// ---- POUs/BACnet_FBCode/FB_BACnet_SCSII_2_GRAHA_ENERGY.TcPOU
(* Usage : 
fbSCSII_2_GRAHA_ENERGY : FB_BACnet_SCSII_2_GRAHA_ENERGY :=(Client:=(nDeviceInstance := 356)); 
*)
FUNCTION_BLOCK  FB_BACnet_SCSII_2_GRAHA_ENERGY
VAR_INPUT CONSTANT
	Client : FB_BACnet_Client := (tReadCycleTime:=T#10S,nMaxParallelRequests:=20);
	SCSII_2_GRAHA_ENERGY: FB_BACnetRM_Device := (Client:=Client);
	Exhaust_Fan_GF_1_ST: FB_BACnetRM_BI := (Client:=Client,nObjectInstance:=208);
	Exhaust_Fan_GF_1_TR: FB_BACnetRM_BI := (Client:=Client,nObjectInstance:=209);
	Exhaust_Fan_GF_2_ST: FB_BACnetRM_BI := (Client:=Client,nObjectInstance:=210);
	Exhaust_Fan_GF_2_TR: FB_BACnetRM_BI := (Client:=Client,nObjectInstance:=211);
	Exhaust_Fan_GF_3_ST: FB_BACnetRM_BI := (Client:=Client,nObjectInstance:=212);
	Exhaust_Fan_GF_3_TR: FB_BACnetRM_BI := (Client:=Client,nObjectInstance:=213);
	Intake_Fan_GF_1_ST: FB_BACnetRM_BI := (Client:=Client,nObjectInstance:=214);
	Intake_Fan_GF_1_TR: FB_BACnetRM_BI := (Client:=Client,nObjectInstance:=215);
	Intake_Fan_GF_2_ST: FB_BACnetRM_BI := (Client:=Client,nObjectInstance:=216);
	Intake_Fan_GF_2_TR: FB_BACnetRM_BI := (Client:=Client,nObjectInstance:=217);
	Toilet_Exh_Fan_GF_1_ST: FB_BACnetRM_BI := (Client:=Client,nObjectInstance:=218);
	Toilet_Exh_Fan_GF_1_TR: FB_BACnetRM_BI := (Client:=Client,nObjectInstance:=219);
	Exhaust_Fan_MZ_1_ST: FB_BACnetRM_BI := (Client:=Client,nObjectInstance:=220);
	Exhaust_Fan_MZ_1_TR: FB_BACnetRM_BI := (Client:=Client,nObjectInstance:=221);
	Exhaust_Fan_MZ_2_ST: FB_BACnetRM_BI := (Client:=Client,nObjectInstance:=222);
	Exhaust_Fan_MZ_2_TR: FB_BACnetRM_BI := (Client:=Client,nObjectInstance:=223);
	Exhaust_Fan_MZ_3_ST: FB_BACnetRM_BI := (Client:=Client,nObjectInstance:=224);
	Exhaust_Fan_MZ_3_TR: FB_BACnetRM_BI := (Client:=Client,nObjectInstance:=225);
	Exhaust_Fan_MZ_4_ST: FB_BACnetRM_BI := (Client:=Client,nObjectInstance:=226);
	Exhaust_Fan_MZ_4_TR: FB_BACnetRM_BI := (Client:=Client,nObjectInstance:=227);
	Exhaust_Fan_MZ_5_ST: FB_BACnetRM_BI := (Client:=Client,nObjectInstance:=228);
	Exhaust_Fan_MZ_5_TR: FB_BACnetRM_BI := (Client:=Client,nObjectInstance:=229);
	Exhaust_Fan_MZ_6_ST: FB_BACnetRM_BI := (Client:=Client,nObjectInstance:=230);
	Exhaust_Fan_MZ_6_TR: FB_BACnetRM_BI := (Client:=Client,nObjectInstance:=231);
	Exhaust_Fan_MZ_7_ST: FB_BACnetRM_BI := (Client:=Client,nObjectInstance:=232);
	Exhaust_Fan_MZ_7_TR: FB_BACnetRM_BI := (Client:=Client,nObjectInstance:=233);
	Intake_Fan_MZ_1_ST: FB_BACnetRM_BI := (Client:=Client,nObjectInstance:=234);
	Intake_Fan_MZ_1_TR: FB_BACnetRM_BI := (Client:=Client,nObjectInstance:=235);
	Toilet_Exh_Fan_MZ_1_ST: FB_BACnetRM_BI := (Client:=Client,nObjectInstance:=236);
	Toilet_Exh_Fan_MZ_1_TR: FB_BACnetRM_BI := (Client:=Client,nObjectInstance:=237);
	Exhaust_Fan_2_1_ST: FB_BACnetRM_BI := (Client:=Client,nObjectInstance:=238);
	Exhaust_Fan_2_1_TR: FB_BACnetRM_BI := (Client:=Client,nObjectInstance:=239);
	Exhaust_Fan_2_2_ST: FB_BACnetRM_BI := (Client:=Client,nObjectInstance:=240);
	Exhaust_Fan_2_2_TR: FB_BACnetRM_BI := (Client:=Client,nObjectInstance:=241);
	Exhaust_Fan_2_3_ST: FB_BACnetRM_BI := (Client:=Client,nObjectInstance:=242);
	Exhaust_Fan_2_3_TR: FB_BACnetRM_BI := (Client:=Client,nObjectInstance:=243);
	Exhaust_Fan_2_4_ST: FB_BACnetRM_BI := (Client:=Client,nObjectInstance:=244);
	Exhaust_Fan_2_4_TR: FB_BACnetRM_BI := (Client:=Client,nObjectInstance:=245);
	Intake_Fan_2_1_ST: FB_BACnetRM_BI := (Client:=Client,nObjectInstance:=246);
	Intake_Fan_2_1_TR: FB_BACnetRM_BI := (Client:=Client,nObjectInstance:=247);
	Intake_Fan_2_2_ST: FB_BACnetRM_BI := (Client:=Client,nObjectInstance:=248);
	Intake_Fan_2_2_TR: FB_BACnetRM_BI := (Client:=Client,nObjectInstance:=249);
	Intake_Fan_2_3_ST: FB_BACnetRM_BI := (Client:=Client,nObjectInstance:=250);
	Intake_Fan_2_3_TR: FB_BACnetRM_BI := (Client:=Client,nObjectInstance:=251);
	Toilet_Exh_Fan_2_1_ST: FB_BACnetRM_BI := (Client:=Client,nObjectInstance:=252);
	Toilet_Exh_Fan_2_1_TR: FB_BACnetRM_BI := (Client:=Client,nObjectInstance:=253);
	Intake_Fan_4_1_ST: FB_BACnetRM_BI := (Client:=Client,nObjectInstance:=254);
	Intake_Fan_4_1_TR: FB_BACnetRM_BI := (Client:=Client,nObjectInstance:=255);
	Intake_Fan_4_2_ST: FB_BACnetRM_BI := (Client:=Client,nObjectInstance:=256);
	Intake_Fan_4_2_TR: FB_BACnetRM_BI := (Client:=Client,nObjectInstance:=257);
	Intake_Fan_4_3_ST: FB_BACnetRM_BI := (Client:=Client,nObjectInstance:=258);
	Intake_Fan_4_3_TR: FB_BACnetRM_BI := (Client:=Client,nObjectInstance:=259);
	Exhaust_Fan_4_5_ST: FB_BACnetRM_BI := (Client:=Client,nObjectInstance:=260);
	Exhaust_Fan_4_5_TR: FB_BACnetRM_BI := (Client:=Client,nObjectInstance:=261);
	Exhaust_Fan_4_6_ST: FB_BACnetRM_BI := (Client:=Client,nObjectInstance:=262);
	Exhaust_Fan_4_6_TR: FB_BACnetRM_BI := (Client:=Client,nObjectInstance:=263);
	Exhaust_Fan_4_7_ST: FB_BACnetRM_BI := (Client:=Client,nObjectInstance:=264);
	Exhaust_Fan_4_7_TR: FB_BACnetRM_BI := (Client:=Client,nObjectInstance:=265);
	Exhaust_Fan_3_7_ST: FB_BACnetRM_BI := (Client:=Client,nObjectInstance:=266);
	Exhaust_Fan_3_7_TR: FB_BACnetRM_BI := (Client:=Client,nObjectInstance:=267);
	Intake_Fan_3_1_ST: FB_BACnetRM_BI := (Client:=Client,nObjectInstance:=268);
	General_Fire_Alm: FB_BACnetRM_BI := (Client:=Client,nObjectInstance:=269);
	Intake_Fan_3_2_ST: FB_BACnetRM_BI := (Client:=Client,nObjectInstance:=270);
	Intake_Fan_3_2_TR: FB_BACnetRM_BI := (Client:=Client,nObjectInstance:=271);
	Exhaust_Fan_B5_1_ST: FB_BACnetRM_BI := (Client:=Client,nObjectInstance:=470);
	Exhaust_Fan_B5_2_ST: FB_BACnetRM_BI := (Client:=Client,nObjectInstance:=471);
	Exhaust_Fan_B5_3_ST: FB_BACnetRM_BI := (Client:=Client,nObjectInstance:=472);
	Intake_Fan_B5_1_ST: FB_BACnetRM_BI := (Client:=Client,nObjectInstance:=473);
	Intake_Fan_B5_2_ST: FB_BACnetRM_BI := (Client:=Client,nObjectInstance:=474);
	Intake_Fan_B5_3_ST: FB_BACnetRM_BI := (Client:=Client,nObjectInstance:=475);
	Spare_1_ST: FB_BACnetRM_BI := (Client:=Client,nObjectInstance:=476);
	Spare_2_ST: FB_BACnetRM_BI := (Client:=Client,nObjectInstance:=477);
	Exhaust_Fan_B5_1_TR: FB_BACnetRM_BI := (Client:=Client,nObjectInstance:=478);
	Exhaust_Fan_B5_2_TR: FB_BACnetRM_BI := (Client:=Client,nObjectInstance:=479);
	Exhaust_Fan_B5_3_TR: FB_BACnetRM_BI := (Client:=Client,nObjectInstance:=480);
	Intake_Fan_B5_1_TR: FB_BACnetRM_BI := (Client:=Client,nObjectInstance:=481);
	Intake_Fan_B5_2_TR: FB_BACnetRM_BI := (Client:=Client,nObjectInstance:=482);
	Intake_Fan_B5_3_TR: FB_BACnetRM_BI := (Client:=Client,nObjectInstance:=483);
	Spare_1_TR: FB_BACnetRM_BI := (Client:=Client,nObjectInstance:=484);
	Spare_2_TR: FB_BACnetRM_BI := (Client:=Client,nObjectInstance:=485);
	Exhaust_Fan_B4_1_ST: FB_BACnetRM_BI := (Client:=Client,nObjectInstance:=486);
	Exhaust_Fan_B4_2_ST: FB_BACnetRM_BI := (Client:=Client,nObjectInstance:=487);
	Exhaust_Fan_B4_3_ST: FB_BACnetRM_BI := (Client:=Client,nObjectInstance:=488);
	Intake_Fan_B4_1_ST: FB_BACnetRM_BI := (Client:=Client,nObjectInstance:=489);
	Intake_Fan_B4_2_ST: FB_BACnetRM_BI := (Client:=Client,nObjectInstance:=490);
	Intake_Fan_B4_3_ST: FB_BACnetRM_BI := (Client:=Client,nObjectInstance:=491);
	Spare_1_ST_X: FB_BACnetRM_BI := (Client:=Client,nObjectInstance:=492);
	Spare_2_ST_X: FB_BACnetRM_BI := (Client:=Client,nObjectInstance:=493);
	Exhaust_Fan_B4_1_TR: FB_BACnetRM_BI := (Client:=Client,nObjectInstance:=494);
	Exhaust_Fan_B4_2_TR: FB_BACnetRM_BI := (Client:=Client,nObjectInstance:=495);
	Exhaust_Fan_B4_3_TR: FB_BACnetRM_BI := (Client:=Client,nObjectInstance:=496);
	Intake_Fan_B4_1_TR: FB_BACnetRM_BI := (Client:=Client,nObjectInstance:=497);
	Intake_Fan_B4_2_TR: FB_BACnetRM_BI := (Client:=Client,nObjectInstance:=498);
	Intake_Fan_B4_3_TR: FB_BACnetRM_BI := (Client:=Client,nObjectInstance:=499);
	Spare_1_TR_X: FB_BACnetRM_BI := (Client:=Client,nObjectInstance:=500);
	Spare_2_TR_X: FB_BACnetRM_BI := (Client:=Client,nObjectInstance:=501);
	Exhaust_Fan_B3_1_ST: FB_BACnetRM_BI := (Client:=Client,nObjectInstance:=502);
	Exhaust_Fan_B3_2_ST: FB_BACnetRM_BI := (Client:=Client,nObjectInstance:=503);
	Exhaust_Fan_B3_3_ST: FB_BACnetRM_BI := (Client:=Client,nObjectInstance:=504);
	Intake_Fan_B3_1_ST: FB_BACnetRM_BI := (Client:=Client,nObjectInstance:=505);
	Intake_Fan_B3_2_ST: FB_BACnetRM_BI := (Client:=Client,nObjectInstance:=506);
	Intake_Fan_B3_3_ST: FB_BACnetRM_BI := (Client:=Client,nObjectInstance:=507);
	Spare_1_ST_X_X: FB_BACnetRM_BI := (Client:=Client,nObjectInstance:=508);
	Spare_2_ST_X_X: FB_BACnetRM_BI := (Client:=Client,nObjectInstance:=509);
	Exhaust_Fan_B3_1_TR: FB_BACnetRM_BI := (Client:=Client,nObjectInstance:=510);
	Exhaust_Fan_B3_2_TR: FB_BACnetRM_BI := (Client:=Client,nObjectInstance:=511);
	Exhaust_Fan_B3_3_TR: FB_BACnetRM_BI := (Client:=Client,nObjectInstance:=512);
	Intake_Fan_B3_1_TR: FB_BACnetRM_BI := (Client:=Client,nObjectInstance:=513);
	Intake_Fan_B3_2_TR: FB_BACnetRM_BI := (Client:=Client,nObjectInstance:=514);
	Intake_Fan_B3_3_TR: FB_BACnetRM_BI := (Client:=Client,nObjectInstance:=515);
	Spare_1_TR_X_X: FB_BACnetRM_BI := (Client:=Client,nObjectInstance:=516);
	Spare_2_TR_X_X: FB_BACnetRM_BI := (Client:=Client,nObjectInstance:=517);
	Exhaust_Fan_B2_1_ST: FB_BACnetRM_BI := (Client:=Client,nObjectInstance:=518);
	Exhaust_Fan_B2_2_ST: FB_BACnetRM_BI := (Client:=Client,nObjectInstance:=519);
	Exhaust_Fan_B2_3_ST: FB_BACnetRM_BI := (Client:=Client,nObjectInstance:=520);
	Intake_Fan_B2_1_ST: FB_BACnetRM_BI := (Client:=Client,nObjectInstance:=521);
	Intake_Fan_B2_2_ST: FB_BACnetRM_BI := (Client:=Client,nObjectInstance:=522);
	Intake_Fan_B2_3_ST: FB_BACnetRM_BI := (Client:=Client,nObjectInstance:=523);
	Reset_Alarm_Fire_Pump_S: FB_BACnetRM_BI := (Client:=Client,nObjectInstance:=524);
	Spare_2_ST_X_X_X: FB_BACnetRM_BI := (Client:=Client,nObjectInstance:=525);
	Exhaust_Fan_B2_1_TR: FB_BACnetRM_BI := (Client:=Client,nObjectInstance:=526);
	Exhaust_Fan_B2_2_TR: FB_BACnetRM_BI := (Client:=Client,nObjectInstance:=527);
	Exhaust_Fan_B2_3_TR: FB_BACnetRM_BI := (Client:=Client,nObjectInstance:=528);
	Intake_Fan_B2_1_TR: FB_BACnetRM_BI := (Client:=Client,nObjectInstance:=529);
	Intake_Fan_B2_2_TR: FB_BACnetRM_BI := (Client:=Client,nObjectInstance:=530);
	Intake_Fan_B2_3_TR: FB_BACnetRM_BI := (Client:=Client,nObjectInstance:=531);
	Spare_1_TR_X_X_X: FB_BACnetRM_BI := (Client:=Client,nObjectInstance:=532);
	Spare_2_TR_X_X_X: FB_BACnetRM_BI := (Client:=Client,nObjectInstance:=533);
	Exhaust_Fan_B1_1_ST: FB_BACnetRM_BI := (Client:=Client,nObjectInstance:=534);
	Exhaust_Fan_B1_2_ST: FB_BACnetRM_BI := (Client:=Client,nObjectInstance:=535);
	Exhaust_Fan_B1_3_ST: FB_BACnetRM_BI := (Client:=Client,nObjectInstance:=536);
	Intake_Fan_B1_1_ST: FB_BACnetRM_BI := (Client:=Client,nObjectInstance:=537);
	Intake_Fan_B1_2_ST: FB_BACnetRM_BI := (Client:=Client,nObjectInstance:=538);
	Intake_Fan_B1_3_ST: FB_BACnetRM_BI := (Client:=Client,nObjectInstance:=539);
	Spare_1_ST_X_X_X: FB_BACnetRM_BI := (Client:=Client,nObjectInstance:=540);
	Spare_2_ST_X_X_X_X: FB_BACnetRM_BI := (Client:=Client,nObjectInstance:=541);
	Exhaust_Fan_B1_1_TR: FB_BACnetRM_BI := (Client:=Client,nObjectInstance:=542);
	Exhaust_Fan_B1_2_TR: FB_BACnetRM_BI := (Client:=Client,nObjectInstance:=543);
	Exhaust_Fan_B1_3_TR: FB_BACnetRM_BI := (Client:=Client,nObjectInstance:=544);
	Intake_Fan_B1_1_TR: FB_BACnetRM_BI := (Client:=Client,nObjectInstance:=545);
	Intake_Fan_B1_2_TR: FB_BACnetRM_BI := (Client:=Client,nObjectInstance:=546);
	Intake_Fan_B1_3_TR: FB_BACnetRM_BI := (Client:=Client,nObjectInstance:=547);
	Spare_1_TR_X_X_X_X: FB_BACnetRM_BI := (Client:=Client,nObjectInstance:=548);
	Spare_2_TR_X_X_X_X: FB_BACnetRM_BI := (Client:=Client,nObjectInstance:=549);
	Intake_Fan_3_3_ST: FB_BACnetRM_BI := (Client:=Client,nObjectInstance:=599);
	Intake_Fan_3_3_TR: FB_BACnetRM_BI := (Client:=Client,nObjectInstance:=600);
	Toilet_Exh_Fan_3_1_ST: FB_BACnetRM_BI := (Client:=Client,nObjectInstance:=601);
	Toilet_Exh_Fan_3_1_TR: FB_BACnetRM_BI := (Client:=Client,nObjectInstance:=602);
	Exh_Fan_Mech_2_1_ST: FB_BACnetRM_BI := (Client:=Client,nObjectInstance:=603);
	Exh_Fan_Mech_2_2_ST: FB_BACnetRM_BI := (Client:=Client,nObjectInstance:=604);
	Exh_Fan_Mech_2_1_TR: FB_BACnetRM_BI := (Client:=Client,nObjectInstance:=605);
	Exh_Fan_Mech_2_2_TR: FB_BACnetRM_BI := (Client:=Client,nObjectInstance:=606);
	Exh_Fan_Mech_3_ST: FB_BACnetRM_BI := (Client:=Client,nObjectInstance:=607);
	Exh_Fan_Mech_3_TR: FB_BACnetRM_BI := (Client:=Client,nObjectInstance:=608);
	Press_Fan_Mech_3_ST: FB_BACnetRM_BI := (Client:=Client,nObjectInstance:=609);
	Press_Fan_Mech_3_TR: FB_BACnetRM_BI := (Client:=Client,nObjectInstance:=610);
	Press_Fan_1_Mech_3_1_ST: FB_BACnetRM_BI := (Client:=Client,nObjectInstance:=611);
	Press_Fan_1_Mech_3_1_TR: FB_BACnetRM_BI := (Client:=Client,nObjectInstance:=612);
	Press_Fan_2_Mech_3_2_ST: FB_BACnetRM_BI := (Client:=Client,nObjectInstance:=613);
	Press_Fan_2_Mech_3_2_TR: FB_BACnetRM_BI := (Client:=Client,nObjectInstance:=614);
	Press_Fan_3_Mech_3_3_ST: FB_BACnetRM_BI := (Client:=Client,nObjectInstance:=615);
	Press_Fan_3_Mech_3_3_TR: FB_BACnetRM_BI := (Client:=Client,nObjectInstance:=616);
	CHILLER_1_ST: FB_BACnetRM_BI := (Client:=Client,nObjectInstance:=625);
	CHILLER_1_TR: FB_BACnetRM_BI := (Client:=Client,nObjectInstance:=626);
	CHILLER_2_ST: FB_BACnetRM_BI := (Client:=Client,nObjectInstance:=627);
	CHILLER_2_TR: FB_BACnetRM_BI := (Client:=Client,nObjectInstance:=628);
	CHILLER_3_ST: FB_BACnetRM_BI := (Client:=Client,nObjectInstance:=629);
	CHILLER_3_TR: FB_BACnetRM_BI := (Client:=Client,nObjectInstance:=630);
	CHILLER_4_ST: FB_BACnetRM_BI := (Client:=Client,nObjectInstance:=631);
	CHILLER_4_TR: FB_BACnetRM_BI := (Client:=Client,nObjectInstance:=632);
	CHWP_1_ST: FB_BACnetRM_BI := (Client:=Client,nObjectInstance:=633);
	CHWP_1_TR: FB_BACnetRM_BI := (Client:=Client,nObjectInstance:=634);
	CHWP_2_ST: FB_BACnetRM_BI := (Client:=Client,nObjectInstance:=635);
	CHWP_2_TR: FB_BACnetRM_BI := (Client:=Client,nObjectInstance:=636);
	CHWP_3_ST: FB_BACnetRM_BI := (Client:=Client,nObjectInstance:=637);
	CHWP_3_TR: FB_BACnetRM_BI := (Client:=Client,nObjectInstance:=638);
	CHWP_4_ST: FB_BACnetRM_BI := (Client:=Client,nObjectInstance:=639);
	CHWP_4_TR: FB_BACnetRM_BI := (Client:=Client,nObjectInstance:=640);
	AHU_1_ST: FB_BACnetRM_BI := (Client:=Client,nObjectInstance:=641);
	AHU_1TR: FB_BACnetRM_BI := (Client:=Client,nObjectInstance:=642);
	FS_CHILLER_1: FB_BACnetRM_BI := (Client:=Client,nObjectInstance:=643);
	FS_CHILLER_2: FB_BACnetRM_BI := (Client:=Client,nObjectInstance:=644);
	FS_CHILLER_3: FB_BACnetRM_BI := (Client:=Client,nObjectInstance:=645);
	FS_CHILLER_4: FB_BACnetRM_BI := (Client:=Client,nObjectInstance:=646);
	DPS_AHU_1: FB_BACnetRM_BI := (Client:=Client,nObjectInstance:=647);
	AFS_AHU_1: FB_BACnetRM_BI := (Client:=Client,nObjectInstance:=648);
	AHU_2_ST: FB_BACnetRM_BI := (Client:=Client,nObjectInstance:=649);
	AHU_2_TR: FB_BACnetRM_BI := (Client:=Client,nObjectInstance:=650);
	DPS_AHU_2: FB_BACnetRM_BI := (Client:=Client,nObjectInstance:=651);
	AFS_AHU_2: FB_BACnetRM_BI := (Client:=Client,nObjectInstance:=652);
	Exh_Fan_Mech_1_ST: FB_BACnetRM_BI := (Client:=Client,nObjectInstance:=653);
	Exh_Fan_Mech_1_TR: FB_BACnetRM_BI := (Client:=Client,nObjectInstance:=654);
	Press_Fan_1_Mech_1_ST: FB_BACnetRM_BI := (Client:=Client,nObjectInstance:=655);
	Press_Fan_1_Mech_1_TR: FB_BACnetRM_BI := (Client:=Client,nObjectInstance:=656);
	Press_Fan_2_Mech_1_ST: FB_BACnetRM_BI := (Client:=Client,nObjectInstance:=657);
	Press_Fan_2_Mech_1_TR: FB_BACnetRM_BI := (Client:=Client,nObjectInstance:=658);
	Press_Fan3_Mech_1_ST: FB_BACnetRM_BI := (Client:=Client,nObjectInstance:=659);
	Press_Fan_3_Mech_1_TR: FB_BACnetRM_BI := (Client:=Client,nObjectInstance:=660);
	Press_Fan_FA_Mech_1_ST: FB_BACnetRM_BI := (Client:=Client,nObjectInstance:=661);
	Press_Fan_FA_Mech_1_TR: FB_BACnetRM_BI := (Client:=Client,nObjectInstance:=662);
	SSP_1A_AUTO_MAN_ST: FB_BACnetRM_BI := (Client:=Client,nObjectInstance:=663);
	SSP_1A_TR: FB_BACnetRM_BI := (Client:=Client,nObjectInstance:=664);
	SSP_1B_AUTO_MAN_ST: FB_BACnetRM_BI := (Client:=Client,nObjectInstance:=665);
	SSP_1B_TR: FB_BACnetRM_BI := (Client:=Client,nObjectInstance:=666);
	SSP_2A_AUTO_MAN_ST: FB_BACnetRM_BI := (Client:=Client,nObjectInstance:=667);
	SSP_2A_TR: FB_BACnetRM_BI := (Client:=Client,nObjectInstance:=668);
	SSP_2B_AUTO_MAN_ST: FB_BACnetRM_BI := (Client:=Client,nObjectInstance:=669);
	SSP_2B_TR: FB_BACnetRM_BI := (Client:=Client,nObjectInstance:=670);
	SSP_3A_AUTO_MAN_ST: FB_BACnetRM_BI := (Client:=Client,nObjectInstance:=671);
	SSP_3A_TR: FB_BACnetRM_BI := (Client:=Client,nObjectInstance:=672);
	SSP_3B_AUTO_MAN_ST: FB_BACnetRM_BI := (Client:=Client,nObjectInstance:=673);
	SSP_3B_TR: FB_BACnetRM_BI := (Client:=Client,nObjectInstance:=674);
	SSP_4A_AUTO_MAN_ST: FB_BACnetRM_BI := (Client:=Client,nObjectInstance:=675);
	SSP_4A_TR: FB_BACnetRM_BI := (Client:=Client,nObjectInstance:=676);
	SSP_4B_AUTO_MAN_ST: FB_BACnetRM_BI := (Client:=Client,nObjectInstance:=677);
	SSP_4B_TR: FB_BACnetRM_BI := (Client:=Client,nObjectInstance:=678);
	DELIVERY_PUMP_1_ON_OF: FB_BACnetRM_BI := (Client:=Client,nObjectInstance:=679);
	DELIVERY_PUMP_2_ON_OF: FB_BACnetRM_BI := (Client:=Client,nObjectInstance:=680);
	DELIVERY_PUMP_1_TR: FB_BACnetRM_BI := (Client:=Client,nObjectInstance:=681);
	DELIVERY_PUMP_2_TR: FB_BACnetRM_BI := (Client:=Client,nObjectInstance:=682);
	DSP_1A_AUTO_MAN_ST: FB_BACnetRM_BI := (Client:=Client,nObjectInstance:=683);
	DSP_1A_TR: FB_BACnetRM_BI := (Client:=Client,nObjectInstance:=684);
	DSP_1B_AUTO_MAN_ST: FB_BACnetRM_BI := (Client:=Client,nObjectInstance:=685);
	DSP_1B_TR: FB_BACnetRM_BI := (Client:=Client,nObjectInstance:=686);
	DSP_2A_AUTO_MAN_ST: FB_BACnetRM_BI := (Client:=Client,nObjectInstance:=687);
	DSP_2A_TR: FB_BACnetRM_BI := (Client:=Client,nObjectInstance:=688);
	DSP_2B_AUTO_MAN_ST: FB_BACnetRM_BI := (Client:=Client,nObjectInstance:=689);
	DSP_2B_TR: FB_BACnetRM_BI := (Client:=Client,nObjectInstance:=690);
	DSP_3A_AUTO_MAN_ST: FB_BACnetRM_BI := (Client:=Client,nObjectInstance:=691);
	DSP_3A_TR: FB_BACnetRM_BI := (Client:=Client,nObjectInstance:=692);
	DSP_3B_AUTO_MAN_ST: FB_BACnetRM_BI := (Client:=Client,nObjectInstance:=693);
	DSP_3B_TR: FB_BACnetRM_BI := (Client:=Client,nObjectInstance:=694);
	DSP_4A_AUTO_MAN_ST: FB_BACnetRM_BI := (Client:=Client,nObjectInstance:=695);
	DSP_4A_TR: FB_BACnetRM_BI := (Client:=Client,nObjectInstance:=696);
	DSP_4B_AUTO_MAN_ST: FB_BACnetRM_BI := (Client:=Client,nObjectInstance:=697);
	DSP_4B_TR: FB_BACnetRM_BI := (Client:=Client,nObjectInstance:=698);
	DSP_5A_AUTO_MAN_ST: FB_BACnetRM_BI := (Client:=Client,nObjectInstance:=699);
	DSP_5A_TR: FB_BACnetRM_BI := (Client:=Client,nObjectInstance:=700);
	DSP_5B_AUTO_MAN_ST: FB_BACnetRM_BI := (Client:=Client,nObjectInstance:=701);
	DSP_5B_TR: FB_BACnetRM_BI := (Client:=Client,nObjectInstance:=702);
	DSP_6A_AUTO_MAN_ST: FB_BACnetRM_BI := (Client:=Client,nObjectInstance:=703);
	DSP_6B_AUTO_MAN_ST: FB_BACnetRM_BI := (Client:=Client,nObjectInstance:=704);
	DSP_6A_TR: FB_BACnetRM_BI := (Client:=Client,nObjectInstance:=705);
	DSP_6B_TR: FB_BACnetRM_BI := (Client:=Client,nObjectInstance:=706);
	BOOSTER_PUMP_1_ON_OFF: FB_BACnetRM_BI := (Client:=Client,nObjectInstance:=707);
	BOOSTER_PUMP_1_TR: FB_BACnetRM_BI := (Client:=Client,nObjectInstance:=708);
	BOOSTER_PUMP_2_ON_OFF: FB_BACnetRM_BI := (Client:=Client,nObjectInstance:=709);
	BOOSTER_PUMP_2_TR: FB_BACnetRM_BI := (Client:=Client,nObjectInstance:=710);
	AHU_x_LOBBY_ST: FB_BACnetRM_BI := (Client:=Client,nObjectInstance:=711);
	AHU_x_LOBBY_TR: FB_BACnetRM_BI := (Client:=Client,nObjectInstance:=712);
	DPS_AHU_LOBBY: FB_BACnetRM_BI := (Client:=Client,nObjectInstance:=713);
	AFS_AHU_LOBBY: FB_BACnetRM_BI := (Client:=Client,nObjectInstance:=714);
	Pompa_Fire_Fighting_Die: FB_BACnetRM_BI := (Client:=Client,nObjectInstance:=715);
	Pompa_Fire_Fighting_Ele: FB_BACnetRM_BI := (Client:=Client,nObjectInstance:=716);
	Pompa_Fire_Fighting_Ele_X: FB_BACnetRM_BI := (Client:=Client,nObjectInstance:=717);
	Pompa_Fire_Fighting_Dis: FB_BACnetRM_BI := (Client:=Client,nObjectInstance:=718);
	Pompa_Fire_Fighting_Ele_X_X: FB_BACnetRM_BI := (Client:=Client,nObjectInstance:=719);
	Pompa_Fire_Fighting_Ele_X_X_X: FB_BACnetRM_BI := (Client:=Client,nObjectInstance:=720);
	Pompa_Fire_Fighting_Dis_X: FB_BACnetRM_BI := (Client:=Client,nObjectInstance:=721);
	Pompa_Fire_Fighting_Ele_X_X_X_X: FB_BACnetRM_BI := (Client:=Client,nObjectInstance:=722);
	Pompa_Fire_Fighting_Ele_X_X_X_X_X: FB_BACnetRM_BI := (Client:=Client,nObjectInstance:=723);
	CH_1_SUPP_TEMP: FB_BACnetRM_AI := (Client:=Client,nObjectInstance:=102);
	CH_1_RET_TEMP: FB_BACnetRM_AI := (Client:=Client,nObjectInstance:=103);
	CH_2_SUPP_TEMP: FB_BACnetRM_AI := (Client:=Client,nObjectInstance:=104);
	CH_2_RET_TEMP: FB_BACnetRM_AI := (Client:=Client,nObjectInstance:=105);
	CH_3_SUPP_TEMP: FB_BACnetRM_AI := (Client:=Client,nObjectInstance:=106);
	CH_3_RET_TEMP: FB_BACnetRM_AI := (Client:=Client,nObjectInstance:=107);
	CH_4_SUPP_TEMP: FB_BACnetRM_AI := (Client:=Client,nObjectInstance:=108);
	CH_4_RET_TEMP: FB_BACnetRM_AI := (Client:=Client,nObjectInstance:=109);
	HEADER_SUPP_TEMP: FB_BACnetRM_AI := (Client:=Client,nObjectInstance:=110);
	HEADER_RET_TEMP: FB_BACnetRM_AI := (Client:=Client,nObjectInstance:=111);
	FLOWMETER: FB_BACnetRM_AI := (Client:=Client,nObjectInstance:=112);
	PRESSURE: FB_BACnetRM_AI := (Client:=Client,nObjectInstance:=113);
	PRA_x_3: FB_BACnetRM_AI := (Client:=Client,nObjectInstance:=114);
	PRA_x_4: FB_BACnetRM_AI := (Client:=Client,nObjectInstance:=115);
	PRA_x_5: FB_BACnetRM_AI := (Client:=Client,nObjectInstance:=116);
	PRA_x_6: FB_BACnetRM_AI := (Client:=Client,nObjectInstance:=117);
	PRA_x_7: FB_BACnetRM_AI := (Client:=Client,nObjectInstance:=118);
	PRA_x_8: FB_BACnetRM_AI := (Client:=Client,nObjectInstance:=119);
	PRA_x_9: FB_BACnetRM_AI := (Client:=Client,nObjectInstance:=120);
	PRA_x_10: FB_BACnetRM_AI := (Client:=Client,nObjectInstance:=121);
	AHU_1_SUPP_TEMP: FB_BACnetRM_AI := (Client:=Client,nObjectInstance:=122);
	AHU_1_RET_TEMP: FB_BACnetRM_AI := (Client:=Client,nObjectInstance:=123);
	SUPP_TEMP: FB_BACnetRM_AI := (Client:=Client,nObjectInstance:=124);
	RET_TEMP: FB_BACnetRM_AI := (Client:=Client,nObjectInstance:=125);
	ROOF_WATER_TANK_1_HIGH: FB_BACnetRM_AI := (Client:=Client,nObjectInstance:=126);
	ROOF_WATER_TANK_2_HIGH: FB_BACnetRM_AI := (Client:=Client,nObjectInstance:=127);
	ROOF_WATER_TANK_1_VOLUM: FB_BACnetRM_AI := (Client:=Client,nObjectInstance:=128);
	ROOF_WATER_TANK_2_VOLUM: FB_BACnetRM_AI := (Client:=Client,nObjectInstance:=129);
	SUPP_TEMP_AHU_LOBBY: FB_BACnetRM_AI := (Client:=Client,nObjectInstance:=130);
	RET_TEMP_AHU_LOBBY: FB_BACnetRM_AI := (Client:=Client,nObjectInstance:=131);
	Water_Level_1: FB_BACnetRM_AI := (Client:=Client,nObjectInstance:=132);
	Water_Level_2: FB_BACnetRM_AI := (Client:=Client,nObjectInstance:=133);
	Water_Level_3: FB_BACnetRM_AI := (Client:=Client,nObjectInstance:=134);
	DAILY_TANK: FB_BACnetRM_AI := (Client:=Client,nObjectInstance:=135);
	STORAGE_ABC: FB_BACnetRM_AI := (Client:=Client,nObjectInstance:=136);
	STORAGE_DEF: FB_BACnetRM_AI := (Client:=Client,nObjectInstance:=137);
	Pseudo_Water_Level_1: FB_BACnetRM_AI := (Client:=Client,nObjectInstance:=138);
	Pseudo_Water_Level_2: FB_BACnetRM_AI := (Client:=Client,nObjectInstance:=139);
	Pseudo_Water_Level_3: FB_BACnetRM_AI := (Client:=Client,nObjectInstance:=140);
	Pseudo_Daily_Tank: FB_BACnetRM_AI := (Client:=Client,nObjectInstance:=141);
	Pseudo_Storage_A: FB_BACnetRM_AI := (Client:=Client,nObjectInstance:=142);
	Pseudo_Storage_B: FB_BACnetRM_AI := (Client:=Client,nObjectInstance:=143);
	Pseudo_Storage_C: FB_BACnetRM_AI := (Client:=Client,nObjectInstance:=144);
	Pseudo_Storage_D: FB_BACnetRM_AI := (Client:=Client,nObjectInstance:=145);
	Pseudo_Storage_E: FB_BACnetRM_AI := (Client:=Client,nObjectInstance:=146);
	Pseudo_Storage_F: FB_BACnetRM_AI := (Client:=Client,nObjectInstance:=147);
	Pseudo_Spare_1: FB_BACnetRM_AI := (Client:=Client,nObjectInstance:=148);
	Pseudo_Spare_2: FB_BACnetRM_AI := (Client:=Client,nObjectInstance:=149);
	Pseudo_Spare_3: FB_BACnetRM_AI := (Client:=Client,nObjectInstance:=150);
	Exhaust_Fan_GF_1_S_S: FB_BACnetRM_BO := (Client:=Client,nObjectInstance:=104);
	Exhaust_Fan_GF_2_S_S: FB_BACnetRM_BO := (Client:=Client,nObjectInstance:=105);
	Exhaust_Fan_GF_3_S_S: FB_BACnetRM_BO := (Client:=Client,nObjectInstance:=106);
	Intake_Fan_GF_1_S_S: FB_BACnetRM_BO := (Client:=Client,nObjectInstance:=107);
	Intake_Fan_GF_2_S_S: FB_BACnetRM_BO := (Client:=Client,nObjectInstance:=108);
	Toilet_Exh_Fan_GF_1_S_S: FB_BACnetRM_BO := (Client:=Client,nObjectInstance:=109);
	Exhaust_Fan_MZ_1_S_S: FB_BACnetRM_BO := (Client:=Client,nObjectInstance:=110);
	Exhaust_Fan_MZ_2_S_S: FB_BACnetRM_BO := (Client:=Client,nObjectInstance:=111);
	Exhaust_Fan_MZ_3_S_S: FB_BACnetRM_BO := (Client:=Client,nObjectInstance:=112);
	Exhaust_Fan_MZ_4_S_S: FB_BACnetRM_BO := (Client:=Client,nObjectInstance:=113);
	Exhaust_Fan_MZ_5_S_S: FB_BACnetRM_BO := (Client:=Client,nObjectInstance:=114);
	Exhaust_Fan_MZ_6_S_S: FB_BACnetRM_BO := (Client:=Client,nObjectInstance:=115);
	Exhaust_Fan_MZ_7_S_S: FB_BACnetRM_BO := (Client:=Client,nObjectInstance:=116);
	Intake_Fan_MZ_1_S_S: FB_BACnetRM_BO := (Client:=Client,nObjectInstance:=117);
	Toilet_Exh_Fan_MZ_1_S_S: FB_BACnetRM_BO := (Client:=Client,nObjectInstance:=118);
	Exhaust_Fan_2_1_S_S: FB_BACnetRM_BO := (Client:=Client,nObjectInstance:=119);
	Exhaust_Fan_2_2_S_S: FB_BACnetRM_BO := (Client:=Client,nObjectInstance:=120);
	Exhaust_Fan_2_3_S_S: FB_BACnetRM_BO := (Client:=Client,nObjectInstance:=121);
	Exhaust_Fan_2_4_S_S: FB_BACnetRM_BO := (Client:=Client,nObjectInstance:=122);
	Intake_Fan_2_1_S_S: FB_BACnetRM_BO := (Client:=Client,nObjectInstance:=123);
	Intake_Fan_2_2_S_S: FB_BACnetRM_BO := (Client:=Client,nObjectInstance:=124);
	Intake_Fan_2_3_S_S: FB_BACnetRM_BO := (Client:=Client,nObjectInstance:=125);
	Toilet_Exh_Fan_2_1_S_S: FB_BACnetRM_BO := (Client:=Client,nObjectInstance:=126);
	Intake_Fan_4_1_S_S: FB_BACnetRM_BO := (Client:=Client,nObjectInstance:=127);
	Intake_Fan_4_2_S_S: FB_BACnetRM_BO := (Client:=Client,nObjectInstance:=128);
	Intake_Fan_4_3_S_S: FB_BACnetRM_BO := (Client:=Client,nObjectInstance:=129);
	Exhaust_Fan_4_5_S_S: FB_BACnetRM_BO := (Client:=Client,nObjectInstance:=130);
	Exhaust_Fan_4_6_S_S: FB_BACnetRM_BO := (Client:=Client,nObjectInstance:=131);
	Exhaust_Fan_4_7_S_S: FB_BACnetRM_BO := (Client:=Client,nObjectInstance:=132);
	Exhaust_Fan_3_7_S_S: FB_BACnetRM_BO := (Client:=Client,nObjectInstance:=133);
	Intake_Fan_3_1_S_S: FB_BACnetRM_BO := (Client:=Client,nObjectInstance:=134);
	Intake_Fan_3_2_S_S: FB_BACnetRM_BO := (Client:=Client,nObjectInstance:=135);
	Exhaust_Fan_B5_1_S_S: FB_BACnetRM_BO := (Client:=Client,nObjectInstance:=235);
	Exhaust_Fan_B5_2_S_S: FB_BACnetRM_BO := (Client:=Client,nObjectInstance:=236);
	Exhaust_Fan_B5_3_S_S: FB_BACnetRM_BO := (Client:=Client,nObjectInstance:=237);
	Intake_Fan_B5_1_S_S: FB_BACnetRM_BO := (Client:=Client,nObjectInstance:=238);
	Intake_Fan_B5_2_S_S: FB_BACnetRM_BO := (Client:=Client,nObjectInstance:=239);
	Intake_Fan_B5_3_S_S: FB_BACnetRM_BO := (Client:=Client,nObjectInstance:=240);
	Spare_1_S_S: FB_BACnetRM_BO := (Client:=Client,nObjectInstance:=241);
	Spare_2_S_S: FB_BACnetRM_BO := (Client:=Client,nObjectInstance:=242);
	Exhaust_Fan_B4_1_S_S: FB_BACnetRM_BO := (Client:=Client,nObjectInstance:=243);
	Exhaust_Fan_B4_2_S_S: FB_BACnetRM_BO := (Client:=Client,nObjectInstance:=244);
	Exhaust_Fan_B4_3_S_S: FB_BACnetRM_BO := (Client:=Client,nObjectInstance:=245);
	Intake_Fan_B4_1_S_S: FB_BACnetRM_BO := (Client:=Client,nObjectInstance:=246);
	Intake_Fan_B4_2_S_S: FB_BACnetRM_BO := (Client:=Client,nObjectInstance:=247);
	Intake_Fan_B4_3_S_S: FB_BACnetRM_BO := (Client:=Client,nObjectInstance:=248);
	Spare_1_S_S_X: FB_BACnetRM_BO := (Client:=Client,nObjectInstance:=249);
	Spare_2_S_S_X: FB_BACnetRM_BO := (Client:=Client,nObjectInstance:=250);
	Exhaust_Fan_B3_1_S_S: FB_BACnetRM_BO := (Client:=Client,nObjectInstance:=251);
	Exhaust_Fan_B3_2_S_S: FB_BACnetRM_BO := (Client:=Client,nObjectInstance:=252);
	Exhaust_Fan_B3_3_S_S: FB_BACnetRM_BO := (Client:=Client,nObjectInstance:=253);
	Intake_Fan_B3_1_S_S: FB_BACnetRM_BO := (Client:=Client,nObjectInstance:=254);
	Intake_Fan_B3_2_S_S: FB_BACnetRM_BO := (Client:=Client,nObjectInstance:=255);
	Intake_Fan_B3_3_S_S: FB_BACnetRM_BO := (Client:=Client,nObjectInstance:=256);
	Spare_1_S_S_X_X: FB_BACnetRM_BO := (Client:=Client,nObjectInstance:=257);
	Spare_2_S_S_X_X: FB_BACnetRM_BO := (Client:=Client,nObjectInstance:=258);
	Exhaust_Fan_B2_1_S_S: FB_BACnetRM_BO := (Client:=Client,nObjectInstance:=259);
	Exhaust_Fan_B2_2_S_S: FB_BACnetRM_BO := (Client:=Client,nObjectInstance:=260);
	Exhaust_Fan_B2_3_S_S: FB_BACnetRM_BO := (Client:=Client,nObjectInstance:=261);
	Intake_Fan_B2_1_S_S: FB_BACnetRM_BO := (Client:=Client,nObjectInstance:=262);
	Intake_Fan_B2_2_S_S: FB_BACnetRM_BO := (Client:=Client,nObjectInstance:=263);
	Intake_Fan_B2_3_S_S: FB_BACnetRM_BO := (Client:=Client,nObjectInstance:=264);
	Spare_1_S_S_X_X_X: FB_BACnetRM_BO := (Client:=Client,nObjectInstance:=265);
	Spare_2_S_S_X_X_X: FB_BACnetRM_BO := (Client:=Client,nObjectInstance:=266);
	Exhaust_Fan_B1_1_S_S: FB_BACnetRM_BO := (Client:=Client,nObjectInstance:=267);
	Exhaust_Fan_B1_2_S_S: FB_BACnetRM_BO := (Client:=Client,nObjectInstance:=268);
	Exhaust_Fan_B1_3_S_S: FB_BACnetRM_BO := (Client:=Client,nObjectInstance:=269);
	Intake_Fan_B1_1_S_S: FB_BACnetRM_BO := (Client:=Client,nObjectInstance:=270);
	Intake_Fan_B1_2_S_S: FB_BACnetRM_BO := (Client:=Client,nObjectInstance:=271);
	Intake_Fan_B1_3_S_S: FB_BACnetRM_BO := (Client:=Client,nObjectInstance:=272);
	Spare_1_S_S_X_X_X_X: FB_BACnetRM_BO := (Client:=Client,nObjectInstance:=273);
	Spare_2_S_S_X_X_X_X: FB_BACnetRM_BO := (Client:=Client,nObjectInstance:=274);
	Intake_Fan_3_3_S_S: FB_BACnetRM_BO := (Client:=Client,nObjectInstance:=294);
	Toilet_Exh_Fan_3_1_S_S: FB_BACnetRM_BO := (Client:=Client,nObjectInstance:=295);
	Exh_Fan_Mech_2_1_S_S: FB_BACnetRM_BO := (Client:=Client,nObjectInstance:=296);
	Exh_Fan_Mech_2_2_S_S: FB_BACnetRM_BO := (Client:=Client,nObjectInstance:=297);
	Exh_Fan_Mech_3_S_S: FB_BACnetRM_BO := (Client:=Client,nObjectInstance:=298);
	Press_Fan_Mech_3_S_S: FB_BACnetRM_BO := (Client:=Client,nObjectInstance:=299);
	CHILLER_1_SS: FB_BACnetRM_BO := (Client:=Client,nObjectInstance:=304);
	CHILLER_2_SS: FB_BACnetRM_BO := (Client:=Client,nObjectInstance:=305);
	CHILLER_3_SS: FB_BACnetRM_BO := (Client:=Client,nObjectInstance:=306);
	CHILLER_4_SS: FB_BACnetRM_BO := (Client:=Client,nObjectInstance:=307);
	CHWP_1_SS: FB_BACnetRM_BO := (Client:=Client,nObjectInstance:=308);
	CHWP_2_SS: FB_BACnetRM_BO := (Client:=Client,nObjectInstance:=309);
	CHWP_3_SS: FB_BACnetRM_BO := (Client:=Client,nObjectInstance:=310);
	CHWP_4_SS: FB_BACnetRM_BO := (Client:=Client,nObjectInstance:=311);
	AHU_1_SS: FB_BACnetRM_BO := (Client:=Client,nObjectInstance:=312);
	CH_1_SS: FB_BACnetRM_BO := (Client:=Client,nObjectInstance:=313);
	CH_2_SS: FB_BACnetRM_BO := (Client:=Client,nObjectInstance:=314);
	CH_3_SS: FB_BACnetRM_BO := (Client:=Client,nObjectInstance:=315);
	CH_4_SS: FB_BACnetRM_BO := (Client:=Client,nObjectInstance:=316);
	CH_5_SS: FB_BACnetRM_BO := (Client:=Client,nObjectInstance:=317);
	CH_6_SS: FB_BACnetRM_BO := (Client:=Client,nObjectInstance:=318);
	CH_7_SS: FB_BACnetRM_BO := (Client:=Client,nObjectInstance:=319);
	CH_8_SS: FB_BACnetRM_BO := (Client:=Client,nObjectInstance:=320);
	CH_9_SS: FB_BACnetRM_BO := (Client:=Client,nObjectInstance:=321);
	CH_10_SS: FB_BACnetRM_BO := (Client:=Client,nObjectInstance:=322);
	AHU_2_SS: FB_BACnetRM_BO := (Client:=Client,nObjectInstance:=323);
	SPARE: FB_BACnetRM_BO := (Client:=Client,nObjectInstance:=324);
	Press_Fan_FA_Mech_1_S_S: FB_BACnetRM_BO := (Client:=Client,nObjectInstance:=325);
	Press_Fan_1_Mech_1_S_S: FB_BACnetRM_BO := (Client:=Client,nObjectInstance:=326);
	Exh_Fan_Mech_1_S_S: FB_BACnetRM_BO := (Client:=Client,nObjectInstance:=327);
	AHU_x_LOBBY_SS: FB_BACnetRM_BO := (Client:=Client,nObjectInstance:=328);
	SPARE_X: FB_BACnetRM_BO := (Client:=Client,nObjectInstance:=329);
	ST_Diesel_Pump_Low_Zone: FB_BACnetRM_BO := (Client:=Client,nObjectInstance:=330);
	ST_Elektrik_Pump_Low_Zo: FB_BACnetRM_BO := (Client:=Client,nObjectInstance:=331);
	ALM_Elektrik_Pump_Low_Z: FB_BACnetRM_BO := (Client:=Client,nObjectInstance:=332);
	ST_Diesel_Pump_Medium_Z: FB_BACnetRM_BO := (Client:=Client,nObjectInstance:=333);
	ST_Elektrik_Pump_Medium: FB_BACnetRM_BO := (Client:=Client,nObjectInstance:=334);
	ALM_Elektrik_Pump_Mediu: FB_BACnetRM_BO := (Client:=Client,nObjectInstance:=335);
	ST_Diesel_Pump_High_Zon: FB_BACnetRM_BO := (Client:=Client,nObjectInstance:=336);
	ST_Elektrik_Pump_High_Z: FB_BACnetRM_BO := (Client:=Client,nObjectInstance:=337);
	LM_Elektrik_Pump_High_Z: FB_BACnetRM_BO := (Client:=Client,nObjectInstance:=338);
	MV_AHU: FB_BACnetRM_AO := (Client:=Client,nObjectInstance:=0);
	MV_CHILLER: FB_BACnetRM_AO := (Client:=Client,nObjectInstance:=1);
	SP_RET_TEMP: FB_BACnetRM_AO := (Client:=Client,nObjectInstance:=2);
	SP_SUPP_TEMP: FB_BACnetRM_AO := (Client:=Client,nObjectInstance:=3);
	MV_AHU_2: FB_BACnetRM_AO := (Client:=Client,nObjectInstance:=4);
	SP_RET_TEMP_X: FB_BACnetRM_AO := (Client:=Client,nObjectInstance:=5);
	MV_AHU_LOBBY: FB_BACnetRM_AO := (Client:=Client,nObjectInstance:=6);
	SP_RET_TEMP_AHU_LOBBY: FB_BACnetRM_AO := (Client:=Client,nObjectInstance:=7);
	Pseudo_Spare_4: FB_BACnetRM_AO := (Client:=Client,nObjectInstance:=8);
	Pseudo_Spare_5: FB_BACnetRM_AO := (Client:=Client,nObjectInstance:=9);
	Pseudo_Spare_6: FB_BACnetRM_AO := (Client:=Client,nObjectInstance:=10);
	fire: FB_BACnetRM_MI := (Client:=Client,nObjectInstance:=0);
	pwf: FB_BACnetRM_MI := (Client:=Client,nObjectInstance:=1);
END_VAR

Client();
SCSII_2_GRAHA_ENERGY();
Exhaust_Fan_GF_1_ST();
Exhaust_Fan_GF_1_TR();
Exhaust_Fan_GF_2_ST();
Exhaust_Fan_GF_2_TR();
Exhaust_Fan_GF_3_ST();
Exhaust_Fan_GF_3_TR();
Intake_Fan_GF_1_ST();
Intake_Fan_GF_1_TR();
Intake_Fan_GF_2_ST();
Intake_Fan_GF_2_TR();
Toilet_Exh_Fan_GF_1_ST();
Toilet_Exh_Fan_GF_1_TR();
Exhaust_Fan_MZ_1_ST();
Exhaust_Fan_MZ_1_TR();
Exhaust_Fan_MZ_2_ST();
Exhaust_Fan_MZ_2_TR();
Exhaust_Fan_MZ_3_ST();
Exhaust_Fan_MZ_3_TR();
Exhaust_Fan_MZ_4_ST();
Exhaust_Fan_MZ_4_TR();
Exhaust_Fan_MZ_5_ST();
Exhaust_Fan_MZ_5_TR();
Exhaust_Fan_MZ_6_ST();
Exhaust_Fan_MZ_6_TR();
Exhaust_Fan_MZ_7_ST();
Exhaust_Fan_MZ_7_TR();
Intake_Fan_MZ_1_ST();
Intake_Fan_MZ_1_TR();
Toilet_Exh_Fan_MZ_1_ST();
Toilet_Exh_Fan_MZ_1_TR();
Exhaust_Fan_2_1_ST();
Exhaust_Fan_2_1_TR();
Exhaust_Fan_2_2_ST();
Exhaust_Fan_2_2_TR();
Exhaust_Fan_2_3_ST();
Exhaust_Fan_2_3_TR();
Exhaust_Fan_2_4_ST();
Exhaust_Fan_2_4_TR();
Intake_Fan_2_1_ST();
Intake_Fan_2_1_TR();
Intake_Fan_2_2_ST();
Intake_Fan_2_2_TR();
Intake_Fan_2_3_ST();
Intake_Fan_2_3_TR();
Toilet_Exh_Fan_2_1_ST();
Toilet_Exh_Fan_2_1_TR();
Intake_Fan_4_1_ST();
Intake_Fan_4_1_TR();
Intake_Fan_4_2_ST();
Intake_Fan_4_2_TR();
Intake_Fan_4_3_ST();
Intake_Fan_4_3_TR();
Exhaust_Fan_4_5_ST();
Exhaust_Fan_4_5_TR();
Exhaust_Fan_4_6_ST();
Exhaust_Fan_4_6_TR();
Exhaust_Fan_4_7_ST();
Exhaust_Fan_4_7_TR();
Exhaust_Fan_3_7_ST();
Exhaust_Fan_3_7_TR();
Intake_Fan_3_1_ST();
General_Fire_Alm();
Intake_Fan_3_2_ST();
Intake_Fan_3_2_TR();
Exhaust_Fan_B5_1_ST();
Exhaust_Fan_B5_2_ST();
Exhaust_Fan_B5_3_ST();
Intake_Fan_B5_1_ST();
Intake_Fan_B5_2_ST();
Intake_Fan_B5_3_ST();
Spare_1_ST();
Spare_2_ST();
Exhaust_Fan_B5_1_TR();
Exhaust_Fan_B5_2_TR();
Exhaust_Fan_B5_3_TR();
Intake_Fan_B5_1_TR();
Intake_Fan_B5_2_TR();
Intake_Fan_B5_3_TR();
Spare_1_TR();
Spare_2_TR();
Exhaust_Fan_B4_1_ST();
Exhaust_Fan_B4_2_ST();
Exhaust_Fan_B4_3_ST();
Intake_Fan_B4_1_ST();
Intake_Fan_B4_2_ST();
Intake_Fan_B4_3_ST();
Spare_1_ST_X();
Spare_2_ST_X();
Exhaust_Fan_B4_1_TR();
Exhaust_Fan_B4_2_TR();
Exhaust_Fan_B4_3_TR();
Intake_Fan_B4_1_TR();
Intake_Fan_B4_2_TR();
Intake_Fan_B4_3_TR();
Spare_1_TR_X();
Spare_2_TR_X();
Exhaust_Fan_B3_1_ST();
Exhaust_Fan_B3_2_ST();
Exhaust_Fan_B3_3_ST();
Intake_Fan_B3_1_ST();
Intake_Fan_B3_2_ST();
Intake_Fan_B3_3_ST();
Spare_1_ST_X_X();
Spare_2_ST_X_X();
Exhaust_Fan_B3_1_TR();
Exhaust_Fan_B3_2_TR();
Exhaust_Fan_B3_3_TR();
Intake_Fan_B3_1_TR();
Intake_Fan_B3_2_TR();
Intake_Fan_B3_3_TR();
Spare_1_TR_X_X();
Spare_2_TR_X_X();
Exhaust_Fan_B2_1_ST();
Exhaust_Fan_B2_2_ST();
Exhaust_Fan_B2_3_ST();
Intake_Fan_B2_1_ST();
Intake_Fan_B2_2_ST();
Intake_Fan_B2_3_ST();
Reset_Alarm_Fire_Pump_S();
Spare_2_ST_X_X_X();
Exhaust_Fan_B2_1_TR();
Exhaust_Fan_B2_2_TR();
Exhaust_Fan_B2_3_TR();
Intake_Fan_B2_1_TR();
Intake_Fan_B2_2_TR();
Intake_Fan_B2_3_TR();
Spare_1_TR_X_X_X();
Spare_2_TR_X_X_X();
Exhaust_Fan_B1_1_ST();
Exhaust_Fan_B1_2_ST();
Exhaust_Fan_B1_3_ST();
Intake_Fan_B1_1_ST();
Intake_Fan_B1_2_ST();
Intake_Fan_B1_3_ST();
Spare_1_ST_X_X_X();
Spare_2_ST_X_X_X_X();
Exhaust_Fan_B1_1_TR();
Exhaust_Fan_B1_2_TR();
Exhaust_Fan_B1_3_TR();
Intake_Fan_B1_1_TR();
Intake_Fan_B1_2_TR();
Intake_Fan_B1_3_TR();
Spare_1_TR_X_X_X_X();
Spare_2_TR_X_X_X_X();
Intake_Fan_3_3_ST();
Intake_Fan_3_3_TR();
Toilet_Exh_Fan_3_1_ST();
Toilet_Exh_Fan_3_1_TR();
Exh_Fan_Mech_2_1_ST();
Exh_Fan_Mech_2_2_ST();
Exh_Fan_Mech_2_1_TR();
Exh_Fan_Mech_2_2_TR();
Exh_Fan_Mech_3_ST();
Exh_Fan_Mech_3_TR();
Press_Fan_Mech_3_ST();
Press_Fan_Mech_3_TR();
Press_Fan_1_Mech_3_1_ST();
Press_Fan_1_Mech_3_1_TR();
Press_Fan_2_Mech_3_2_ST();
Press_Fan_2_Mech_3_2_TR();
Press_Fan_3_Mech_3_3_ST();
Press_Fan_3_Mech_3_3_TR();
CHILLER_1_ST();
CHILLER_1_TR();
CHILLER_2_ST();
CHILLER_2_TR();
CHILLER_3_ST();
CHILLER_3_TR();
CHILLER_4_ST();
CHILLER_4_TR();
CHWP_1_ST();
CHWP_1_TR();
CHWP_2_ST();
CHWP_2_TR();
CHWP_3_ST();
CHWP_3_TR();
CHWP_4_ST();
CHWP_4_TR();
AHU_1_ST();
AHU_1TR();
FS_CHILLER_1();
FS_CHILLER_2();
FS_CHILLER_3();
FS_CHILLER_4();
DPS_AHU_1();
AFS_AHU_1();
AHU_2_ST();
AHU_2_TR();
DPS_AHU_2();
AFS_AHU_2();
Exh_Fan_Mech_1_ST();
Exh_Fan_Mech_1_TR();
Press_Fan_1_Mech_1_ST();
Press_Fan_1_Mech_1_TR();
Press_Fan_2_Mech_1_ST();
Press_Fan_2_Mech_1_TR();
Press_Fan3_Mech_1_ST();
Press_Fan_3_Mech_1_TR();
Press_Fan_FA_Mech_1_ST();
Press_Fan_FA_Mech_1_TR();
SSP_1A_AUTO_MAN_ST();
SSP_1A_TR();
SSP_1B_AUTO_MAN_ST();
SSP_1B_TR();
SSP_2A_AUTO_MAN_ST();
SSP_2A_TR();
SSP_2B_AUTO_MAN_ST();
SSP_2B_TR();
SSP_3A_AUTO_MAN_ST();
SSP_3A_TR();
SSP_3B_AUTO_MAN_ST();
SSP_3B_TR();
SSP_4A_AUTO_MAN_ST();
SSP_4A_TR();
SSP_4B_AUTO_MAN_ST();
SSP_4B_TR();
DELIVERY_PUMP_1_ON_OF();
DELIVERY_PUMP_2_ON_OF();
DELIVERY_PUMP_1_TR();
DELIVERY_PUMP_2_TR();
DSP_1A_AUTO_MAN_ST();
DSP_1A_TR();
DSP_1B_AUTO_MAN_ST();
DSP_1B_TR();
DSP_2A_AUTO_MAN_ST();
DSP_2A_TR();
DSP_2B_AUTO_MAN_ST();
DSP_2B_TR();
DSP_3A_AUTO_MAN_ST();
DSP_3A_TR();
DSP_3B_AUTO_MAN_ST();
DSP_3B_TR();
DSP_4A_AUTO_MAN_ST();
DSP_4A_TR();
DSP_4B_AUTO_MAN_ST();
DSP_4B_TR();
DSP_5A_AUTO_MAN_ST();
DSP_5A_TR();
DSP_5B_AUTO_MAN_ST();
DSP_5B_TR();
DSP_6A_AUTO_MAN_ST();
DSP_6B_AUTO_MAN_ST();
DSP_6A_TR();
DSP_6B_TR();
BOOSTER_PUMP_1_ON_OFF();
BOOSTER_PUMP_1_TR();
BOOSTER_PUMP_2_ON_OFF();
BOOSTER_PUMP_2_TR();
AHU_x_LOBBY_ST();
AHU_x_LOBBY_TR();
DPS_AHU_LOBBY();
AFS_AHU_LOBBY();
Pompa_Fire_Fighting_Die();
Pompa_Fire_Fighting_Ele();
Pompa_Fire_Fighting_Ele_X();
Pompa_Fire_Fighting_Dis();
Pompa_Fire_Fighting_Ele_X_X();
Pompa_Fire_Fighting_Ele_X_X_X();
Pompa_Fire_Fighting_Dis_X();
Pompa_Fire_Fighting_Ele_X_X_X_X();
Pompa_Fire_Fighting_Ele_X_X_X_X_X();
CH_1_SUPP_TEMP();
CH_1_RET_TEMP();
CH_2_SUPP_TEMP();
CH_2_RET_TEMP();
CH_3_SUPP_TEMP();
CH_3_RET_TEMP();
CH_4_SUPP_TEMP();
CH_4_RET_TEMP();
HEADER_SUPP_TEMP();
HEADER_RET_TEMP();
FLOWMETER();
PRESSURE();
PRA_x_3();
PRA_x_4();
PRA_x_5();
PRA_x_6();
PRA_x_7();
PRA_x_8();
PRA_x_9();
PRA_x_10();
AHU_1_SUPP_TEMP();
AHU_1_RET_TEMP();
SUPP_TEMP();
RET_TEMP();
ROOF_WATER_TANK_1_HIGH();
ROOF_WATER_TANK_2_HIGH();
ROOF_WATER_TANK_1_VOLUM();
ROOF_WATER_TANK_2_VOLUM();
SUPP_TEMP_AHU_LOBBY();
RET_TEMP_AHU_LOBBY();
Water_Level_1();
Water_Level_2();
Water_Level_3();
DAILY_TANK();
STORAGE_ABC();
STORAGE_DEF();
Pseudo_Water_Level_1();
Pseudo_Water_Level_2();
Pseudo_Water_Level_3();
Pseudo_Daily_Tank();
Pseudo_Storage_A();
Pseudo_Storage_B();
Pseudo_Storage_C();
Pseudo_Storage_D();
Pseudo_Storage_E();
Pseudo_Storage_F();
Pseudo_Spare_1();
Pseudo_Spare_2();
Pseudo_Spare_3();
Exhaust_Fan_GF_1_S_S();
Exhaust_Fan_GF_2_S_S();
Exhaust_Fan_GF_3_S_S();
Intake_Fan_GF_1_S_S();
Intake_Fan_GF_2_S_S();
Toilet_Exh_Fan_GF_1_S_S();
Exhaust_Fan_MZ_1_S_S();
Exhaust_Fan_MZ_2_S_S();
Exhaust_Fan_MZ_3_S_S();
Exhaust_Fan_MZ_4_S_S();
Exhaust_Fan_MZ_5_S_S();
Exhaust_Fan_MZ_6_S_S();
Exhaust_Fan_MZ_7_S_S();
Intake_Fan_MZ_1_S_S();
Toilet_Exh_Fan_MZ_1_S_S();
Exhaust_Fan_2_1_S_S();
Exhaust_Fan_2_2_S_S();
Exhaust_Fan_2_3_S_S();
Exhaust_Fan_2_4_S_S();
Intake_Fan_2_1_S_S();
Intake_Fan_2_2_S_S();
Intake_Fan_2_3_S_S();
Toilet_Exh_Fan_2_1_S_S();
Intake_Fan_4_1_S_S();
Intake_Fan_4_2_S_S();
Intake_Fan_4_3_S_S();
Exhaust_Fan_4_5_S_S();
Exhaust_Fan_4_6_S_S();
Exhaust_Fan_4_7_S_S();
Exhaust_Fan_3_7_S_S();
Intake_Fan_3_1_S_S();
Intake_Fan_3_2_S_S();
Exhaust_Fan_B5_1_S_S();
Exhaust_Fan_B5_2_S_S();
Exhaust_Fan_B5_3_S_S();
Intake_Fan_B5_1_S_S();
Intake_Fan_B5_2_S_S();
Intake_Fan_B5_3_S_S();
Spare_1_S_S();
Spare_2_S_S();
Exhaust_Fan_B4_1_S_S();
Exhaust_Fan_B4_2_S_S();
Exhaust_Fan_B4_3_S_S();
Intake_Fan_B4_1_S_S();
Intake_Fan_B4_2_S_S();
Intake_Fan_B4_3_S_S();
Spare_1_S_S_X();
Spare_2_S_S_X();
Exhaust_Fan_B3_1_S_S();
Exhaust_Fan_B3_2_S_S();
Exhaust_Fan_B3_3_S_S();
Intake_Fan_B3_1_S_S();
Intake_Fan_B3_2_S_S();
Intake_Fan_B3_3_S_S();
Spare_1_S_S_X_X();
Spare_2_S_S_X_X();
Exhaust_Fan_B2_1_S_S();
Exhaust_Fan_B2_2_S_S();
Exhaust_Fan_B2_3_S_S();
Intake_Fan_B2_1_S_S();
Intake_Fan_B2_2_S_S();
Intake_Fan_B2_3_S_S();
Spare_1_S_S_X_X_X();
Spare_2_S_S_X_X_X();
Exhaust_Fan_B1_1_S_S();
Exhaust_Fan_B1_2_S_S();
Exhaust_Fan_B1_3_S_S();
Intake_Fan_B1_1_S_S();
Intake_Fan_B1_2_S_S();
Intake_Fan_B1_3_S_S();
Spare_1_S_S_X_X_X_X();
Spare_2_S_S_X_X_X_X();
Intake_Fan_3_3_S_S();
Toilet_Exh_Fan_3_1_S_S();
Exh_Fan_Mech_2_1_S_S();
Exh_Fan_Mech_2_2_S_S();
Exh_Fan_Mech_3_S_S();
Press_Fan_Mech_3_S_S();
CHILLER_1_SS();
CHILLER_2_SS();
CHILLER_3_SS();
CHILLER_4_SS();
CHWP_1_SS();
CHWP_2_SS();
CHWP_3_SS();
CHWP_4_SS();
AHU_1_SS();
CH_1_SS();
CH_2_SS();
CH_3_SS();
CH_4_SS();
CH_5_SS();
CH_6_SS();
CH_7_SS();
CH_8_SS();
CH_9_SS();
CH_10_SS();
AHU_2_SS();
SPARE();
Press_Fan_FA_Mech_1_S_S();
Press_Fan_1_Mech_1_S_S();
Exh_Fan_Mech_1_S_S();
AHU_x_LOBBY_SS();
SPARE_X();
ST_Diesel_Pump_Low_Zone();
ST_Elektrik_Pump_Low_Zo();
ALM_Elektrik_Pump_Low_Z();
ST_Diesel_Pump_Medium_Z();
ST_Elektrik_Pump_Medium();
ALM_Elektrik_Pump_Mediu();
ST_Diesel_Pump_High_Zon();
ST_Elektrik_Pump_High_Z();
LM_Elektrik_Pump_High_Z();
MV_AHU();
MV_CHILLER();
SP_RET_TEMP();
SP_SUPP_TEMP();
MV_AHU_2();
SP_RET_TEMP_X();
MV_AHU_LOBBY();
SP_RET_TEMP_AHU_LOBBY();
Pseudo_Spare_4();
Pseudo_Spare_5();
Pseudo_Spare_6();
fire();
pwf();

END_FUNCTION_BLOCK

// ---- POUs/BACnet_FBCode/FB_BACnet_DAIKIN_MasterStation_III_No_1.TcPOU
(* Usage : 
fbDAIKIN_MasterStation_III_No_1 : FB_BACnet_DAIKIN_MasterStation_III_No_1 :=(Client:=(nDeviceInstance := 1)); 
*)
FUNCTION_BLOCK  FB_BACnet_DAIKIN_MasterStation_III_No_1
VAR_INPUT CONSTANT
	Client : FB_BACnet_Client := (tReadCycleTime:=T#10S,nMaxParallelRequests:=20);
	DAIKIN_MasterStation_III_No_1: FB_BACnetRM_Device := (Client:=Client);
	StartStopCommand_000: FB_BACnetRM_BO := (Client:=Client,nObjectInstance:=1);
	StartStopStatus_000: FB_BACnetRM_BI := (Client:=Client,nObjectInstance:=2);
	Alarm_000: FB_BACnetRM_BI := (Client:=Client,nObjectInstance:=3);
	MalfunctionCode_000: FB_BACnetRM_MI := (Client:=Client,nObjectInstance:=4);
	
	
	
	
	RoomTemp_000: FB_BACnetRM_AI := (Client:=Client,nObjectInstance:=9);
	TempAdjust_000: FB_BACnetRM_AV := (Client:=Client,nObjectInstance:=10);
	FilterSign_000: FB_BACnetRM_BI := (Client:=Client,nObjectInstance:=11);
	FilterSignReset_000: FB_BACnetRM_BV := (Client:=Client,nObjectInstance:=12);
	RemoteControlStart_000: FB_BACnetRM_BV := (Client:=Client,nObjectInstance:=13);
	
	RemoteControlTempAdjust_000: FB_BACnetRM_BV := (Client:=Client,nObjectInstance:=16);
	
	
	
	
	
	
	
	
	
	
	
	
	StartStopCommand_001: FB_BACnetRM_BO := (Client:=Client,nObjectInstance:=257);
	StartStopStatus_001: FB_BACnetRM_BI := (Client:=Client,nObjectInstance:=258);
	Alarm_001: FB_BACnetRM_BI := (Client:=Client,nObjectInstance:=259);
	MalfunctionCode_001: FB_BACnetRM_MI := (Client:=Client,nObjectInstance:=260);
	
	
	
	
	RoomTemp_001: FB_BACnetRM_AI := (Client:=Client,nObjectInstance:=265);
	TempAdjust_001: FB_BACnetRM_AV := (Client:=Client,nObjectInstance:=266);
	FilterSign_001: FB_BACnetRM_BI := (Client:=Client,nObjectInstance:=267);
	FilterSignReset_001: FB_BACnetRM_BV := (Client:=Client,nObjectInstance:=268);
	RemoteControlStart_001: FB_BACnetRM_BV := (Client:=Client,nObjectInstance:=269);
	
	RemoteControlTempAdjust_001: FB_BACnetRM_BV := (Client:=Client,nObjectInstance:=272);
	
	
	
	
	
	
	
	
	
	
	
	
	StartStopCommand_002: FB_BACnetRM_BO := (Client:=Client,nObjectInstance:=513);
	StartStopStatus_002: FB_BACnetRM_BI := (Client:=Client,nObjectInstance:=514);
	Alarm_002: FB_BACnetRM_BI := (Client:=Client,nObjectInstance:=515);
	MalfunctionCode_002: FB_BACnetRM_MI := (Client:=Client,nObjectInstance:=516);
	
	
	
	
	RoomTemp_002: FB_BACnetRM_AI := (Client:=Client,nObjectInstance:=521);
	TempAdjust_002: FB_BACnetRM_AV := (Client:=Client,nObjectInstance:=522);
	FilterSign_002: FB_BACnetRM_BI := (Client:=Client,nObjectInstance:=523);
	FilterSignReset_002: FB_BACnetRM_BV := (Client:=Client,nObjectInstance:=524);
	RemoteControlStart_002: FB_BACnetRM_BV := (Client:=Client,nObjectInstance:=525);
	
	RemoteControlTempAdjust_002: FB_BACnetRM_BV := (Client:=Client,nObjectInstance:=528);
	
	
	
	
	
	
	
	
	
	
	
	
	StartStopCommand_003: FB_BACnetRM_BO := (Client:=Client,nObjectInstance:=769);
	StartStopStatus_003: FB_BACnetRM_BI := (Client:=Client,nObjectInstance:=770);
	Alarm_003: FB_BACnetRM_BI := (Client:=Client,nObjectInstance:=771);
	MalfunctionCode_003: FB_BACnetRM_MI := (Client:=Client,nObjectInstance:=772);
	
	
	
	
	RoomTemp_003: FB_BACnetRM_AI := (Client:=Client,nObjectInstance:=777);
	TempAdjust_003: FB_BACnetRM_AV := (Client:=Client,nObjectInstance:=778);
	FilterSign_003: FB_BACnetRM_BI := (Client:=Client,nObjectInstance:=779);
	FilterSignReset_003: FB_BACnetRM_BV := (Client:=Client,nObjectInstance:=780);
	RemoteControlStart_003: FB_BACnetRM_BV := (Client:=Client,nObjectInstance:=781);
	
	RemoteControlTempAdjust_003: FB_BACnetRM_BV := (Client:=Client,nObjectInstance:=784);
	
	
	
	
	
	
	
	
	
	
	
	
	StartStopCommand_004: FB_BACnetRM_BO := (Client:=Client,nObjectInstance:=1025);
	StartStopStatus_004: FB_BACnetRM_BI := (Client:=Client,nObjectInstance:=1026);
	Alarm_004: FB_BACnetRM_BI := (Client:=Client,nObjectInstance:=1027);
	MalfunctionCode_004: FB_BACnetRM_MI := (Client:=Client,nObjectInstance:=1028);
	
	
	
	
	RoomTemp_004: FB_BACnetRM_AI := (Client:=Client,nObjectInstance:=1033);
	TempAdjust_004: FB_BACnetRM_AV := (Client:=Client,nObjectInstance:=1034);
	FilterSign_004: FB_BACnetRM_BI := (Client:=Client,nObjectInstance:=1035);
	FilterSignReset_004: FB_BACnetRM_BV := (Client:=Client,nObjectInstance:=1036);
	RemoteControlStart_004: FB_BACnetRM_BV := (Client:=Client,nObjectInstance:=1037);
	
	RemoteControlTempAdjust_004: FB_BACnetRM_BV := (Client:=Client,nObjectInstance:=1040);
	
	
	
	
	
	
	
	
	
	
	
	
	StartStopCommand_005: FB_BACnetRM_BO := (Client:=Client,nObjectInstance:=1281);
	StartStopStatus_005: FB_BACnetRM_BI := (Client:=Client,nObjectInstance:=1282);
	Alarm_005: FB_BACnetRM_BI := (Client:=Client,nObjectInstance:=1283);
	MalfunctionCode_005: FB_BACnetRM_MI := (Client:=Client,nObjectInstance:=1284);
	
	
	
	
	RoomTemp_005: FB_BACnetRM_AI := (Client:=Client,nObjectInstance:=1289);
	TempAdjust_005: FB_BACnetRM_AV := (Client:=Client,nObjectInstance:=1290);
	FilterSign_005: FB_BACnetRM_BI := (Client:=Client,nObjectInstance:=1291);
	FilterSignReset_005: FB_BACnetRM_BV := (Client:=Client,nObjectInstance:=1292);
	RemoteControlStart_005: FB_BACnetRM_BV := (Client:=Client,nObjectInstance:=1293);
	
	RemoteControlTempAdjust_005: FB_BACnetRM_BV := (Client:=Client,nObjectInstance:=1296);
	
	
	
	
	
	
	
	
	
	
	
	
	StartStopCommand_006: FB_BACnetRM_BO := (Client:=Client,nObjectInstance:=1537);
	StartStopStatus_006: FB_BACnetRM_BI := (Client:=Client,nObjectInstance:=1538);
	Alarm_006: FB_BACnetRM_BI := (Client:=Client,nObjectInstance:=1539);
	MalfunctionCode_006: FB_BACnetRM_MI := (Client:=Client,nObjectInstance:=1540);
	
	
	
	
	RoomTemp_006: FB_BACnetRM_AI := (Client:=Client,nObjectInstance:=1545);
	TempAdjust_006: FB_BACnetRM_AV := (Client:=Client,nObjectInstance:=1546);
	FilterSign_006: FB_BACnetRM_BI := (Client:=Client,nObjectInstance:=1547);
	FilterSignReset_006: FB_BACnetRM_BV := (Client:=Client,nObjectInstance:=1548);
	RemoteControlStart_006: FB_BACnetRM_BV := (Client:=Client,nObjectInstance:=1549);
	
	RemoteControlTempAdjust_006: FB_BACnetRM_BV := (Client:=Client,nObjectInstance:=1552);
	
	
	
	
	
	
	
	
	
	
	
	
	StartStopCommand_007: FB_BACnetRM_BO := (Client:=Client,nObjectInstance:=1793);
	StartStopStatus_007: FB_BACnetRM_BI := (Client:=Client,nObjectInstance:=1794);
	Alarm_007: FB_BACnetRM_BI := (Client:=Client,nObjectInstance:=1795);
	MalfunctionCode_007: FB_BACnetRM_MI := (Client:=Client,nObjectInstance:=1796);
	
	
	
	
	RoomTemp_007: FB_BACnetRM_AI := (Client:=Client,nObjectInstance:=1801);
	TempAdjust_007: FB_BACnetRM_AV := (Client:=Client,nObjectInstance:=1802);
	FilterSign_007: FB_BACnetRM_BI := (Client:=Client,nObjectInstance:=1803);
	FilterSignReset_007: FB_BACnetRM_BV := (Client:=Client,nObjectInstance:=1804);
	RemoteControlStart_007: FB_BACnetRM_BV := (Client:=Client,nObjectInstance:=1805);
	
	RemoteControlTempAdjust_007: FB_BACnetRM_BV := (Client:=Client,nObjectInstance:=1808);
	
	
	
	
	
	
	
	
	
	
	
	
	StartStopCommand_008: FB_BACnetRM_BO := (Client:=Client,nObjectInstance:=2049);
	StartStopStatus_008: FB_BACnetRM_BI := (Client:=Client,nObjectInstance:=2050);
	Alarm_008: FB_BACnetRM_BI := (Client:=Client,nObjectInstance:=2051);
	MalfunctionCode_008: FB_BACnetRM_MI := (Client:=Client,nObjectInstance:=2052);
	
	
	
	
	RoomTemp_008: FB_BACnetRM_AI := (Client:=Client,nObjectInstance:=2057);
	TempAdjust_008: FB_BACnetRM_AV := (Client:=Client,nObjectInstance:=2058);
	FilterSign_008: FB_BACnetRM_BI := (Client:=Client,nObjectInstance:=2059);
	FilterSignReset_008: FB_BACnetRM_BV := (Client:=Client,nObjectInstance:=2060);
	RemoteControlStart_008: FB_BACnetRM_BV := (Client:=Client,nObjectInstance:=2061);
	
	RemoteControlTempAdjust_008: FB_BACnetRM_BV := (Client:=Client,nObjectInstance:=2064);
	
	
	
	
	
	
	
	
	
	
	
	
	StartStopCommand_009: FB_BACnetRM_BO := (Client:=Client,nObjectInstance:=2305);
	StartStopStatus_009: FB_BACnetRM_BI := (Client:=Client,nObjectInstance:=2306);
	Alarm_009: FB_BACnetRM_BI := (Client:=Client,nObjectInstance:=2307);
	MalfunctionCode_009: FB_BACnetRM_MI := (Client:=Client,nObjectInstance:=2308);
	
	
	
	
	RoomTemp_009: FB_BACnetRM_AI := (Client:=Client,nObjectInstance:=2313);
	TempAdjust_009: FB_BACnetRM_AV := (Client:=Client,nObjectInstance:=2314);
	FilterSign_009: FB_BACnetRM_BI := (Client:=Client,nObjectInstance:=2315);
	FilterSignReset_009: FB_BACnetRM_BV := (Client:=Client,nObjectInstance:=2316);
	RemoteControlStart_009: FB_BACnetRM_BV := (Client:=Client,nObjectInstance:=2317);
	
	RemoteControlTempAdjust_009: FB_BACnetRM_BV := (Client:=Client,nObjectInstance:=2320);
	
	
	
	
	
	
	
	
	
	
	
	
	StartStopCommand_010: FB_BACnetRM_BO := (Client:=Client,nObjectInstance:=2561);
	StartStopStatus_010: FB_BACnetRM_BI := (Client:=Client,nObjectInstance:=2562);
	Alarm_010: FB_BACnetRM_BI := (Client:=Client,nObjectInstance:=2563);
	MalfunctionCode_010: FB_BACnetRM_MI := (Client:=Client,nObjectInstance:=2564);
	
	
	
	
	RoomTemp_010: FB_BACnetRM_AI := (Client:=Client,nObjectInstance:=2569);
	TempAdjust_010: FB_BACnetRM_AV := (Client:=Client,nObjectInstance:=2570);
	FilterSign_010: FB_BACnetRM_BI := (Client:=Client,nObjectInstance:=2571);
	FilterSignReset_010: FB_BACnetRM_BV := (Client:=Client,nObjectInstance:=2572);
	RemoteControlStart_010: FB_BACnetRM_BV := (Client:=Client,nObjectInstance:=2573);
	
	RemoteControlTempAdjust_010: FB_BACnetRM_BV := (Client:=Client,nObjectInstance:=2576);
	
	
	
	
	
	
	
	
	
	
	
	
	StartStopCommand_011: FB_BACnetRM_BO := (Client:=Client,nObjectInstance:=2817);
	StartStopStatus_011: FB_BACnetRM_BI := (Client:=Client,nObjectInstance:=2818);
	Alarm_011: FB_BACnetRM_BI := (Client:=Client,nObjectInstance:=2819);
	MalfunctionCode_011: FB_BACnetRM_MI := (Client:=Client,nObjectInstance:=2820);
	
	
	
	
	RoomTemp_011: FB_BACnetRM_AI := (Client:=Client,nObjectInstance:=2825);
	TempAdjust_011: FB_BACnetRM_AV := (Client:=Client,nObjectInstance:=2826);
	FilterSign_011: FB_BACnetRM_BI := (Client:=Client,nObjectInstance:=2827);
	FilterSignReset_011: FB_BACnetRM_BV := (Client:=Client,nObjectInstance:=2828);
	RemoteControlStart_011: FB_BACnetRM_BV := (Client:=Client,nObjectInstance:=2829);
	
	RemoteControlTempAdjust_011: FB_BACnetRM_BV := (Client:=Client,nObjectInstance:=2832);
	
	
	
	
	
	
	
	
	
	
	
	
	StartStopCommand_012: FB_BACnetRM_BO := (Client:=Client,nObjectInstance:=3073);
	StartStopStatus_012: FB_BACnetRM_BI := (Client:=Client,nObjectInstance:=3074);
	Alarm_012: FB_BACnetRM_BI := (Client:=Client,nObjectInstance:=3075);
	MalfunctionCode_012: FB_BACnetRM_MI := (Client:=Client,nObjectInstance:=3076);
	
	
	
	
	RoomTemp_012: FB_BACnetRM_AI := (Client:=Client,nObjectInstance:=3081);
	TempAdjust_012: FB_BACnetRM_AV := (Client:=Client,nObjectInstance:=3082);
	FilterSign_012: FB_BACnetRM_BI := (Client:=Client,nObjectInstance:=3083);
	FilterSignReset_012: FB_BACnetRM_BV := (Client:=Client,nObjectInstance:=3084);
	RemoteControlStart_012: FB_BACnetRM_BV := (Client:=Client,nObjectInstance:=3085);
	
	RemoteControlTempAdjust_012: FB_BACnetRM_BV := (Client:=Client,nObjectInstance:=3088);
	
	
	
	
	
	
	
	
	
	
	
	
	StartStopCommand_013: FB_BACnetRM_BO := (Client:=Client,nObjectInstance:=3329);
	StartStopStatus_013: FB_BACnetRM_BI := (Client:=Client,nObjectInstance:=3330);
	Alarm_013: FB_BACnetRM_BI := (Client:=Client,nObjectInstance:=3331);
	MalfunctionCode_013: FB_BACnetRM_MI := (Client:=Client,nObjectInstance:=3332);
	
	
	
	
	RoomTemp_013: FB_BACnetRM_AI := (Client:=Client,nObjectInstance:=3337);
	TempAdjust_013: FB_BACnetRM_AV := (Client:=Client,nObjectInstance:=3338);
	FilterSign_013: FB_BACnetRM_BI := (Client:=Client,nObjectInstance:=3339);
	FilterSignReset_013: FB_BACnetRM_BV := (Client:=Client,nObjectInstance:=3340);
	RemoteControlStart_013: FB_BACnetRM_BV := (Client:=Client,nObjectInstance:=3341);
	
	RemoteControlTempAdjust_013: FB_BACnetRM_BV := (Client:=Client,nObjectInstance:=3344);
	
	
	
	
	
	
	
	
	
	
	
	
	StartStopCommand_014: FB_BACnetRM_BO := (Client:=Client,nObjectInstance:=3585);
	StartStopStatus_014: FB_BACnetRM_BI := (Client:=Client,nObjectInstance:=3586);
	Alarm_014: FB_BACnetRM_BI := (Client:=Client,nObjectInstance:=3587);
	MalfunctionCode_014: FB_BACnetRM_MI := (Client:=Client,nObjectInstance:=3588);
	
	
	
	
	RoomTemp_014: FB_BACnetRM_AI := (Client:=Client,nObjectInstance:=3593);
	TempAdjust_014: FB_BACnetRM_AV := (Client:=Client,nObjectInstance:=3594);
	FilterSign_014: FB_BACnetRM_BI := (Client:=Client,nObjectInstance:=3595);
	FilterSignReset_014: FB_BACnetRM_BV := (Client:=Client,nObjectInstance:=3596);
	RemoteControlStart_014: FB_BACnetRM_BV := (Client:=Client,nObjectInstance:=3597);
	
	RemoteControlTempAdjust_014: FB_BACnetRM_BV := (Client:=Client,nObjectInstance:=3600);
	
	
	
	
	
	
	
	
	
	
	
	
	StartStopCommand_015: FB_BACnetRM_BO := (Client:=Client,nObjectInstance:=3841);
	StartStopStatus_015: FB_BACnetRM_BI := (Client:=Client,nObjectInstance:=3842);
	Alarm_015: FB_BACnetRM_BI := (Client:=Client,nObjectInstance:=3843);
	MalfunctionCode_015: FB_BACnetRM_MI := (Client:=Client,nObjectInstance:=3844);
	
	
	
	
	RoomTemp_015: FB_BACnetRM_AI := (Client:=Client,nObjectInstance:=3849);
	TempAdjust_015: FB_BACnetRM_AV := (Client:=Client,nObjectInstance:=3850);
	FilterSign_015: FB_BACnetRM_BI := (Client:=Client,nObjectInstance:=3851);
	FilterSignReset_015: FB_BACnetRM_BV := (Client:=Client,nObjectInstance:=3852);
	RemoteControlStart_015: FB_BACnetRM_BV := (Client:=Client,nObjectInstance:=3853);
	
	RemoteControlTempAdjust_015: FB_BACnetRM_BV := (Client:=Client,nObjectInstance:=3856);
	
	
	
	
	
	
	
	
	
	
	
	
	StartStopCommand_016: FB_BACnetRM_BO := (Client:=Client,nObjectInstance:=4097);
	StartStopStatus_016: FB_BACnetRM_BI := (Client:=Client,nObjectInstance:=4098);
	Alarm_016: FB_BACnetRM_BI := (Client:=Client,nObjectInstance:=4099);
	MalfunctionCode_016: FB_BACnetRM_MI := (Client:=Client,nObjectInstance:=4100);
	
	
	
	
	RoomTemp_016: FB_BACnetRM_AI := (Client:=Client,nObjectInstance:=4105);
	TempAdjust_016: FB_BACnetRM_AV := (Client:=Client,nObjectInstance:=4106);
	FilterSign_016: FB_BACnetRM_BI := (Client:=Client,nObjectInstance:=4107);
	FilterSignReset_016: FB_BACnetRM_BV := (Client:=Client,nObjectInstance:=4108);
	RemoteControlStart_016: FB_BACnetRM_BV := (Client:=Client,nObjectInstance:=4109);
	
	RemoteControlTempAdjust_016: FB_BACnetRM_BV := (Client:=Client,nObjectInstance:=4112);
	
	
	
	
	
	
	
	
	
	
	
	
	StartStopCommand_017: FB_BACnetRM_BO := (Client:=Client,nObjectInstance:=4353);
	StartStopStatus_017: FB_BACnetRM_BI := (Client:=Client,nObjectInstance:=4354);
	Alarm_017: FB_BACnetRM_BI := (Client:=Client,nObjectInstance:=4355);
	MalfunctionCode_017: FB_BACnetRM_MI := (Client:=Client,nObjectInstance:=4356);
	
	
	
	
	RoomTemp_017: FB_BACnetRM_AI := (Client:=Client,nObjectInstance:=4361);
	TempAdjust_017: FB_BACnetRM_AV := (Client:=Client,nObjectInstance:=4362);
	FilterSign_017: FB_BACnetRM_BI := (Client:=Client,nObjectInstance:=4363);
	FilterSignReset_017: FB_BACnetRM_BV := (Client:=Client,nObjectInstance:=4364);
	RemoteControlStart_017: FB_BACnetRM_BV := (Client:=Client,nObjectInstance:=4365);
	
	RemoteControlTempAdjust_017: FB_BACnetRM_BV := (Client:=Client,nObjectInstance:=4368);
	
	
	
	
	
	
	
	
	
	
	
	
	StartStopCommand_018: FB_BACnetRM_BO := (Client:=Client,nObjectInstance:=4609);
	StartStopStatus_018: FB_BACnetRM_BI := (Client:=Client,nObjectInstance:=4610);
	Alarm_018: FB_BACnetRM_BI := (Client:=Client,nObjectInstance:=4611);
	MalfunctionCode_018: FB_BACnetRM_MI := (Client:=Client,nObjectInstance:=4612);
	
	
	
	
	RoomTemp_018: FB_BACnetRM_AI := (Client:=Client,nObjectInstance:=4617);
	TempAdjust_018: FB_BACnetRM_AV := (Client:=Client,nObjectInstance:=4618);
	FilterSign_018: FB_BACnetRM_BI := (Client:=Client,nObjectInstance:=4619);
	FilterSignReset_018: FB_BACnetRM_BV := (Client:=Client,nObjectInstance:=4620);
	RemoteControlStart_018: FB_BACnetRM_BV := (Client:=Client,nObjectInstance:=4621);
	
	RemoteControlTempAdjust_018: FB_BACnetRM_BV := (Client:=Client,nObjectInstance:=4624);
	
	
	
	
	
	
	
	
	
	
	
	
	StartStopCommand_019: FB_BACnetRM_BO := (Client:=Client,nObjectInstance:=4865);
	StartStopStatus_019: FB_BACnetRM_BI := (Client:=Client,nObjectInstance:=4866);
	Alarm_019: FB_BACnetRM_BI := (Client:=Client,nObjectInstance:=4867);
	MalfunctionCode_019: FB_BACnetRM_MI := (Client:=Client,nObjectInstance:=4868);
	
	
	
	
	RoomTemp_019: FB_BACnetRM_AI := (Client:=Client,nObjectInstance:=4873);
	TempAdjust_019: FB_BACnetRM_AV := (Client:=Client,nObjectInstance:=4874);
	FilterSign_019: FB_BACnetRM_BI := (Client:=Client,nObjectInstance:=4875);
	FilterSignReset_019: FB_BACnetRM_BV := (Client:=Client,nObjectInstance:=4876);
	RemoteControlStart_019: FB_BACnetRM_BV := (Client:=Client,nObjectInstance:=4877);
	
	RemoteControlTempAdjust_019: FB_BACnetRM_BV := (Client:=Client,nObjectInstance:=4880);
	
	
	
	
	
	
	
	
	
	
	
	
	StartStopCommand_020: FB_BACnetRM_BO := (Client:=Client,nObjectInstance:=5121);
	StartStopStatus_020: FB_BACnetRM_BI := (Client:=Client,nObjectInstance:=5122);
	Alarm_020: FB_BACnetRM_BI := (Client:=Client,nObjectInstance:=5123);
	MalfunctionCode_020: FB_BACnetRM_MI := (Client:=Client,nObjectInstance:=5124);
	
	
	
	
	RoomTemp_020: FB_BACnetRM_AI := (Client:=Client,nObjectInstance:=5129);
	TempAdjust_020: FB_BACnetRM_AV := (Client:=Client,nObjectInstance:=5130);
	FilterSign_020: FB_BACnetRM_BI := (Client:=Client,nObjectInstance:=5131);
	FilterSignReset_020: FB_BACnetRM_BV := (Client:=Client,nObjectInstance:=5132);
	RemoteControlStart_020: FB_BACnetRM_BV := (Client:=Client,nObjectInstance:=5133);
	
	RemoteControlTempAdjust_020: FB_BACnetRM_BV := (Client:=Client,nObjectInstance:=5136);
	
	
	
	
	
	
	
	
	
	
	
	
	StartStopCommand_021: FB_BACnetRM_BO := (Client:=Client,nObjectInstance:=5377);
	StartStopStatus_021: FB_BACnetRM_BI := (Client:=Client,nObjectInstance:=5378);
	Alarm_021: FB_BACnetRM_BI := (Client:=Client,nObjectInstance:=5379);
	MalfunctionCode_021: FB_BACnetRM_MI := (Client:=Client,nObjectInstance:=5380);
	
	
	
	
	RoomTemp_021: FB_BACnetRM_AI := (Client:=Client,nObjectInstance:=5385);
	TempAdjust_021: FB_BACnetRM_AV := (Client:=Client,nObjectInstance:=5386);
	FilterSign_021: FB_BACnetRM_BI := (Client:=Client,nObjectInstance:=5387);
	FilterSignReset_021: FB_BACnetRM_BV := (Client:=Client,nObjectInstance:=5388);
	RemoteControlStart_021: FB_BACnetRM_BV := (Client:=Client,nObjectInstance:=5389);
	
	RemoteControlTempAdjust_021: FB_BACnetRM_BV := (Client:=Client,nObjectInstance:=5392);
	
	
	
	
	
	
	
	
	
	
	
	
	StartStopCommand_022: FB_BACnetRM_BO := (Client:=Client,nObjectInstance:=5633);
	StartStopStatus_022: FB_BACnetRM_BI := (Client:=Client,nObjectInstance:=5634);
	Alarm_022: FB_BACnetRM_BI := (Client:=Client,nObjectInstance:=5635);
	MalfunctionCode_022: FB_BACnetRM_MI := (Client:=Client,nObjectInstance:=5636);
	
	
	
	
	RoomTemp_022: FB_BACnetRM_AI := (Client:=Client,nObjectInstance:=5641);
	TempAdjust_022: FB_BACnetRM_AV := (Client:=Client,nObjectInstance:=5642);
	FilterSign_022: FB_BACnetRM_BI := (Client:=Client,nObjectInstance:=5643);
	FilterSignReset_022: FB_BACnetRM_BV := (Client:=Client,nObjectInstance:=5644);
	RemoteControlStart_022: FB_BACnetRM_BV := (Client:=Client,nObjectInstance:=5645);
	
	RemoteControlTempAdjust_022: FB_BACnetRM_BV := (Client:=Client,nObjectInstance:=5648);
	
	
	
	
	
	
	
	
	
	
	
	
	StartStopCommand_023: FB_BACnetRM_BO := (Client:=Client,nObjectInstance:=5889);
	StartStopStatus_023: FB_BACnetRM_BI := (Client:=Client,nObjectInstance:=5890);
	Alarm_023: FB_BACnetRM_BI := (Client:=Client,nObjectInstance:=5891);
	MalfunctionCode_023: FB_BACnetRM_MI := (Client:=Client,nObjectInstance:=5892);
	
	
	
	
	RoomTemp_023: FB_BACnetRM_AI := (Client:=Client,nObjectInstance:=5897);
	TempAdjust_023: FB_BACnetRM_AV := (Client:=Client,nObjectInstance:=5898);
	FilterSign_023: FB_BACnetRM_BI := (Client:=Client,nObjectInstance:=5899);
	FilterSignReset_023: FB_BACnetRM_BV := (Client:=Client,nObjectInstance:=5900);
	RemoteControlStart_023: FB_BACnetRM_BV := (Client:=Client,nObjectInstance:=5901);
	
	RemoteControlTempAdjust_023: FB_BACnetRM_BV := (Client:=Client,nObjectInstance:=5904);
	
	
	
	
	
	
	
	
	
	
	
	
	StartStopCommand_024: FB_BACnetRM_BO := (Client:=Client,nObjectInstance:=6145);
	StartStopStatus_024: FB_BACnetRM_BI := (Client:=Client,nObjectInstance:=6146);
	Alarm_024: FB_BACnetRM_BI := (Client:=Client,nObjectInstance:=6147);
	MalfunctionCode_024: FB_BACnetRM_MI := (Client:=Client,nObjectInstance:=6148);
	
	
	
	
	RoomTemp_024: FB_BACnetRM_AI := (Client:=Client,nObjectInstance:=6153);
	TempAdjust_024: FB_BACnetRM_AV := (Client:=Client,nObjectInstance:=6154);
	FilterSign_024: FB_BACnetRM_BI := (Client:=Client,nObjectInstance:=6155);
	FilterSignReset_024: FB_BACnetRM_BV := (Client:=Client,nObjectInstance:=6156);
	RemoteControlStart_024: FB_BACnetRM_BV := (Client:=Client,nObjectInstance:=6157);
	
	RemoteControlTempAdjust_024: FB_BACnetRM_BV := (Client:=Client,nObjectInstance:=6160);
	
	
	
	
	
	
	
	
	
	
	
	
	StartStopCommand_025: FB_BACnetRM_BO := (Client:=Client,nObjectInstance:=6401);
	StartStopStatus_025: FB_BACnetRM_BI := (Client:=Client,nObjectInstance:=6402);
	Alarm_025: FB_BACnetRM_BI := (Client:=Client,nObjectInstance:=6403);
	MalfunctionCode_025: FB_BACnetRM_MI := (Client:=Client,nObjectInstance:=6404);
	
	
	
	
	RoomTemp_025: FB_BACnetRM_AI := (Client:=Client,nObjectInstance:=6409);
	TempAdjust_025: FB_BACnetRM_AV := (Client:=Client,nObjectInstance:=6410);
	FilterSign_025: FB_BACnetRM_BI := (Client:=Client,nObjectInstance:=6411);
	FilterSignReset_025: FB_BACnetRM_BV := (Client:=Client,nObjectInstance:=6412);
	RemoteControlStart_025: FB_BACnetRM_BV := (Client:=Client,nObjectInstance:=6413);
	
	RemoteControlTempAdjust_025: FB_BACnetRM_BV := (Client:=Client,nObjectInstance:=6416);
	
	
	
	
	
	
	
	
	
	
	
	
	StartStopCommand_026: FB_BACnetRM_BO := (Client:=Client,nObjectInstance:=6657);
	StartStopStatus_026: FB_BACnetRM_BI := (Client:=Client,nObjectInstance:=6658);
	Alarm_026: FB_BACnetRM_BI := (Client:=Client,nObjectInstance:=6659);
	MalfunctionCode_026: FB_BACnetRM_MI := (Client:=Client,nObjectInstance:=6660);
	
	
	
	
	RoomTemp_026: FB_BACnetRM_AI := (Client:=Client,nObjectInstance:=6665);
	TempAdjust_026: FB_BACnetRM_AV := (Client:=Client,nObjectInstance:=6666);
	FilterSign_026: FB_BACnetRM_BI := (Client:=Client,nObjectInstance:=6667);
	FilterSignReset_026: FB_BACnetRM_BV := (Client:=Client,nObjectInstance:=6668);
	RemoteControlStart_026: FB_BACnetRM_BV := (Client:=Client,nObjectInstance:=6669);
	
	RemoteControlTempAdjust_026: FB_BACnetRM_BV := (Client:=Client,nObjectInstance:=6672);
	
	
	
	
	
	
	
	
	
	
	
	
	StartStopCommand_027: FB_BACnetRM_BO := (Client:=Client,nObjectInstance:=6913);
	StartStopStatus_027: FB_BACnetRM_BI := (Client:=Client,nObjectInstance:=6914);
	Alarm_027: FB_BACnetRM_BI := (Client:=Client,nObjectInstance:=6915);
	MalfunctionCode_027: FB_BACnetRM_MI := (Client:=Client,nObjectInstance:=6916);
	
	
	
	
	RoomTemp_027: FB_BACnetRM_AI := (Client:=Client,nObjectInstance:=6921);
	TempAdjust_027: FB_BACnetRM_AV := (Client:=Client,nObjectInstance:=6922);
	FilterSign_027: FB_BACnetRM_BI := (Client:=Client,nObjectInstance:=6923);
	FilterSignReset_027: FB_BACnetRM_BV := (Client:=Client,nObjectInstance:=6924);
	RemoteControlStart_027: FB_BACnetRM_BV := (Client:=Client,nObjectInstance:=6925);
	
	RemoteControlTempAdjust_027: FB_BACnetRM_BV := (Client:=Client,nObjectInstance:=6928);
	
	
	
	
	
	
	
	
	
	
	
	
	StartStopCommand_028: FB_BACnetRM_BO := (Client:=Client,nObjectInstance:=7169);
	StartStopStatus_028: FB_BACnetRM_BI := (Client:=Client,nObjectInstance:=7170);
	Alarm_028: FB_BACnetRM_BI := (Client:=Client,nObjectInstance:=7171);
	MalfunctionCode_028: FB_BACnetRM_MI := (Client:=Client,nObjectInstance:=7172);
	
	
	
	
	RoomTemp_028: FB_BACnetRM_AI := (Client:=Client,nObjectInstance:=7177);
	TempAdjust_028: FB_BACnetRM_AV := (Client:=Client,nObjectInstance:=7178);
	FilterSign_028: FB_BACnetRM_BI := (Client:=Client,nObjectInstance:=7179);
	FilterSignReset_028: FB_BACnetRM_BV := (Client:=Client,nObjectInstance:=7180);
	RemoteControlStart_028: FB_BACnetRM_BV := (Client:=Client,nObjectInstance:=7181);
	
	RemoteControlTempAdjust_028: FB_BACnetRM_BV := (Client:=Client,nObjectInstance:=7184);
	
	
	
	
	
	
	
	
	
	
	
	
	StartStopCommand_029: FB_BACnetRM_BO := (Client:=Client,nObjectInstance:=7425);
	StartStopStatus_029: FB_BACnetRM_BI := (Client:=Client,nObjectInstance:=7426);
	Alarm_029: FB_BACnetRM_BI := (Client:=Client,nObjectInstance:=7427);
	MalfunctionCode_029: FB_BACnetRM_MI := (Client:=Client,nObjectInstance:=7428);
	
	
	
	
	RoomTemp_029: FB_BACnetRM_AI := (Client:=Client,nObjectInstance:=7433);
	TempAdjust_029: FB_BACnetRM_AV := (Client:=Client,nObjectInstance:=7434);
	FilterSign_029: FB_BACnetRM_BI := (Client:=Client,nObjectInstance:=7435);
	FilterSignReset_029: FB_BACnetRM_BV := (Client:=Client,nObjectInstance:=7436);
	RemoteControlStart_029: FB_BACnetRM_BV := (Client:=Client,nObjectInstance:=7437);
	
	RemoteControlTempAdjust_029: FB_BACnetRM_BV := (Client:=Client,nObjectInstance:=7440);
	
	
	
	
	
	
	
	
	
	
	
	
	StartStopCommand_030: FB_BACnetRM_BO := (Client:=Client,nObjectInstance:=7681);
	StartStopStatus_030: FB_BACnetRM_BI := (Client:=Client,nObjectInstance:=7682);
	Alarm_030: FB_BACnetRM_BI := (Client:=Client,nObjectInstance:=7683);
	MalfunctionCode_030: FB_BACnetRM_MI := (Client:=Client,nObjectInstance:=7684);
	
	
	
	
	RoomTemp_030: FB_BACnetRM_AI := (Client:=Client,nObjectInstance:=7689);
	TempAdjust_030: FB_BACnetRM_AV := (Client:=Client,nObjectInstance:=7690);
	FilterSign_030: FB_BACnetRM_BI := (Client:=Client,nObjectInstance:=7691);
	FilterSignReset_030: FB_BACnetRM_BV := (Client:=Client,nObjectInstance:=7692);
	RemoteControlStart_030: FB_BACnetRM_BV := (Client:=Client,nObjectInstance:=7693);
	
	RemoteControlTempAdjust_030: FB_BACnetRM_BV := (Client:=Client,nObjectInstance:=7696);
	
	
	
	
	
	
	
	
	
	
	
	
	StartStopCommand_031: FB_BACnetRM_BO := (Client:=Client,nObjectInstance:=7937);
	StartStopStatus_031: FB_BACnetRM_BI := (Client:=Client,nObjectInstance:=7938);
	Alarm_031: FB_BACnetRM_BI := (Client:=Client,nObjectInstance:=7939);
	MalfunctionCode_031: FB_BACnetRM_MI := (Client:=Client,nObjectInstance:=7940);
	
	
	
	
	RoomTemp_031: FB_BACnetRM_AI := (Client:=Client,nObjectInstance:=7945);
	TempAdjust_031: FB_BACnetRM_AV := (Client:=Client,nObjectInstance:=7946);
	FilterSign_031: FB_BACnetRM_BI := (Client:=Client,nObjectInstance:=7947);
	FilterSignReset_031: FB_BACnetRM_BV := (Client:=Client,nObjectInstance:=7948);
	RemoteControlStart_031: FB_BACnetRM_BV := (Client:=Client,nObjectInstance:=7949);
	
	RemoteControlTempAdjust_031: FB_BACnetRM_BV := (Client:=Client,nObjectInstance:=7952);
	
	
	
	
	
	
	
	
	
	
	
	
	StartStopCommand_032: FB_BACnetRM_BO := (Client:=Client,nObjectInstance:=8193);
	StartStopStatus_032: FB_BACnetRM_BI := (Client:=Client,nObjectInstance:=8194);
	Alarm_032: FB_BACnetRM_BI := (Client:=Client,nObjectInstance:=8195);
	MalfunctionCode_032: FB_BACnetRM_MI := (Client:=Client,nObjectInstance:=8196);
	
	
	
	
	RoomTemp_032: FB_BACnetRM_AI := (Client:=Client,nObjectInstance:=8201);
	TempAdjust_032: FB_BACnetRM_AV := (Client:=Client,nObjectInstance:=8202);
	FilterSign_032: FB_BACnetRM_BI := (Client:=Client,nObjectInstance:=8203);
	FilterSignReset_032: FB_BACnetRM_BV := (Client:=Client,nObjectInstance:=8204);
	RemoteControlStart_032: FB_BACnetRM_BV := (Client:=Client,nObjectInstance:=8205);
	
	RemoteControlTempAdjust_032: FB_BACnetRM_BV := (Client:=Client,nObjectInstance:=8208);
	
	
	
	
	
	
	
	
	
	
	
	
	StartStopCommand_033: FB_BACnetRM_BO := (Client:=Client,nObjectInstance:=8449);
	StartStopStatus_033: FB_BACnetRM_BI := (Client:=Client,nObjectInstance:=8450);
	Alarm_033: FB_BACnetRM_BI := (Client:=Client,nObjectInstance:=8451);
	MalfunctionCode_033: FB_BACnetRM_MI := (Client:=Client,nObjectInstance:=8452);
	
	
	
	
	RoomTemp_033: FB_BACnetRM_AI := (Client:=Client,nObjectInstance:=8457);
	TempAdjust_033: FB_BACnetRM_AV := (Client:=Client,nObjectInstance:=8458);
	FilterSign_033: FB_BACnetRM_BI := (Client:=Client,nObjectInstance:=8459);
	FilterSignReset_033: FB_BACnetRM_BV := (Client:=Client,nObjectInstance:=8460);
	RemoteControlStart_033: FB_BACnetRM_BV := (Client:=Client,nObjectInstance:=8461);
	
	RemoteControlTempAdjust_033: FB_BACnetRM_BV := (Client:=Client,nObjectInstance:=8464);
	
	
	
	
	
	
	
	
	
	
	
	
	StartStopCommand_034: FB_BACnetRM_BO := (Client:=Client,nObjectInstance:=8705);
	StartStopStatus_034: FB_BACnetRM_BI := (Client:=Client,nObjectInstance:=8706);
	Alarm_034: FB_BACnetRM_BI := (Client:=Client,nObjectInstance:=8707);
	MalfunctionCode_034: FB_BACnetRM_MI := (Client:=Client,nObjectInstance:=8708);
	
	
	
	
	RoomTemp_034: FB_BACnetRM_AI := (Client:=Client,nObjectInstance:=8713);
	TempAdjust_034: FB_BACnetRM_AV := (Client:=Client,nObjectInstance:=8714);
	FilterSign_034: FB_BACnetRM_BI := (Client:=Client,nObjectInstance:=8715);
	FilterSignReset_034: FB_BACnetRM_BV := (Client:=Client,nObjectInstance:=8716);
	RemoteControlStart_034: FB_BACnetRM_BV := (Client:=Client,nObjectInstance:=8717);
	
	RemoteControlTempAdjust_034: FB_BACnetRM_BV := (Client:=Client,nObjectInstance:=8720);
	
	
	
	
	
	
	
	
	
	
	
	
	StartStopCommand_035: FB_BACnetRM_BO := (Client:=Client,nObjectInstance:=8961);
	StartStopStatus_035: FB_BACnetRM_BI := (Client:=Client,nObjectInstance:=8962);
	Alarm_035: FB_BACnetRM_BI := (Client:=Client,nObjectInstance:=8963);
	MalfunctionCode_035: FB_BACnetRM_MI := (Client:=Client,nObjectInstance:=8964);
	
	
	
	
	RoomTemp_035: FB_BACnetRM_AI := (Client:=Client,nObjectInstance:=8969);
	TempAdjust_035: FB_BACnetRM_AV := (Client:=Client,nObjectInstance:=8970);
	FilterSign_035: FB_BACnetRM_BI := (Client:=Client,nObjectInstance:=8971);
	FilterSignReset_035: FB_BACnetRM_BV := (Client:=Client,nObjectInstance:=8972);
	RemoteControlStart_035: FB_BACnetRM_BV := (Client:=Client,nObjectInstance:=8973);
	
	RemoteControlTempAdjust_035: FB_BACnetRM_BV := (Client:=Client,nObjectInstance:=8976);
	
	
	
	
	
	
	
	
	
	
	
	
	StartStopCommand_036: FB_BACnetRM_BO := (Client:=Client,nObjectInstance:=9217);
	StartStopStatus_036: FB_BACnetRM_BI := (Client:=Client,nObjectInstance:=9218);
	Alarm_036: FB_BACnetRM_BI := (Client:=Client,nObjectInstance:=9219);
	MalfunctionCode_036: FB_BACnetRM_MI := (Client:=Client,nObjectInstance:=9220);
	
	
	
	
	RoomTemp_036: FB_BACnetRM_AI := (Client:=Client,nObjectInstance:=9225);
	TempAdjust_036: FB_BACnetRM_AV := (Client:=Client,nObjectInstance:=9226);
	FilterSign_036: FB_BACnetRM_BI := (Client:=Client,nObjectInstance:=9227);
	FilterSignReset_036: FB_BACnetRM_BV := (Client:=Client,nObjectInstance:=9228);
	RemoteControlStart_036: FB_BACnetRM_BV := (Client:=Client,nObjectInstance:=9229);
	
	RemoteControlTempAdjust_036: FB_BACnetRM_BV := (Client:=Client,nObjectInstance:=9232);
	
	
	
	
	
	
	
	
	
	
	
	
	StartStopCommand_037: FB_BACnetRM_BO := (Client:=Client,nObjectInstance:=9473);
	StartStopStatus_037: FB_BACnetRM_BI := (Client:=Client,nObjectInstance:=9474);
	Alarm_037: FB_BACnetRM_BI := (Client:=Client,nObjectInstance:=9475);
	MalfunctionCode_037: FB_BACnetRM_MI := (Client:=Client,nObjectInstance:=9476);
	
	
	
	
	RoomTemp_037: FB_BACnetRM_AI := (Client:=Client,nObjectInstance:=9481);
	TempAdjust_037: FB_BACnetRM_AV := (Client:=Client,nObjectInstance:=9482);
	FilterSign_037: FB_BACnetRM_BI := (Client:=Client,nObjectInstance:=9483);
	FilterSignReset_037: FB_BACnetRM_BV := (Client:=Client,nObjectInstance:=9484);
	RemoteControlStart_037: FB_BACnetRM_BV := (Client:=Client,nObjectInstance:=9485);
	
	RemoteControlTempAdjust_037: FB_BACnetRM_BV := (Client:=Client,nObjectInstance:=9488);
	
	
	
	
	
	
	
	
	
	
	
	
	StartStopCommand_038: FB_BACnetRM_BO := (Client:=Client,nObjectInstance:=9729);
	StartStopStatus_038: FB_BACnetRM_BI := (Client:=Client,nObjectInstance:=9730);
	Alarm_038: FB_BACnetRM_BI := (Client:=Client,nObjectInstance:=9731);
	MalfunctionCode_038: FB_BACnetRM_MI := (Client:=Client,nObjectInstance:=9732);
	
	
	
	
	RoomTemp_038: FB_BACnetRM_AI := (Client:=Client,nObjectInstance:=9737);
	TempAdjust_038: FB_BACnetRM_AV := (Client:=Client,nObjectInstance:=9738);
	FilterSign_038: FB_BACnetRM_BI := (Client:=Client,nObjectInstance:=9739);
	FilterSignReset_038: FB_BACnetRM_BV := (Client:=Client,nObjectInstance:=9740);
	RemoteControlStart_038: FB_BACnetRM_BV := (Client:=Client,nObjectInstance:=9741);
	
	RemoteControlTempAdjust_038: FB_BACnetRM_BV := (Client:=Client,nObjectInstance:=9744);
	
	
	
	
	
	
	
	
	
	
	
	
	StartStopCommand_039: FB_BACnetRM_BO := (Client:=Client,nObjectInstance:=9985);
	StartStopStatus_039: FB_BACnetRM_BI := (Client:=Client,nObjectInstance:=9986);
	Alarm_039: FB_BACnetRM_BI := (Client:=Client,nObjectInstance:=9987);
	MalfunctionCode_039: FB_BACnetRM_MI := (Client:=Client,nObjectInstance:=9988);
	
	
	
	
	RoomTemp_039: FB_BACnetRM_AI := (Client:=Client,nObjectInstance:=9993);
	TempAdjust_039: FB_BACnetRM_AV := (Client:=Client,nObjectInstance:=9994);
	FilterSign_039: FB_BACnetRM_BI := (Client:=Client,nObjectInstance:=9995);
	FilterSignReset_039: FB_BACnetRM_BV := (Client:=Client,nObjectInstance:=9996);
	RemoteControlStart_039: FB_BACnetRM_BV := (Client:=Client,nObjectInstance:=9997);
	
	RemoteControlTempAdjust_039: FB_BACnetRM_BV := (Client:=Client,nObjectInstance:=10000);
	
	
	
	
	
	
	
	
	
	
	
	
	StartStopCommand_041: FB_BACnetRM_BO := (Client:=Client,nObjectInstance:=10497);
	StartStopStatus_041: FB_BACnetRM_BI := (Client:=Client,nObjectInstance:=10498);
	Alarm_041: FB_BACnetRM_BI := (Client:=Client,nObjectInstance:=10499);
	MalfunctionCode_041: FB_BACnetRM_MI := (Client:=Client,nObjectInstance:=10500);
	
	
	
	
	RoomTemp_041: FB_BACnetRM_AI := (Client:=Client,nObjectInstance:=10505);
	TempAdjust_041: FB_BACnetRM_AV := (Client:=Client,nObjectInstance:=10506);
	FilterSign_041: FB_BACnetRM_BI := (Client:=Client,nObjectInstance:=10507);
	FilterSignReset_041: FB_BACnetRM_BV := (Client:=Client,nObjectInstance:=10508);
	RemoteControlStart_041: FB_BACnetRM_BV := (Client:=Client,nObjectInstance:=10509);
	
	RemoteControlTempAdjust_041: FB_BACnetRM_BV := (Client:=Client,nObjectInstance:=10512);
	
	
	
	
	
	
	
	
	
	
	
	
	StartStopCommand_042: FB_BACnetRM_BO := (Client:=Client,nObjectInstance:=10753);
	StartStopStatus_042: FB_BACnetRM_BI := (Client:=Client,nObjectInstance:=10754);
	Alarm_042: FB_BACnetRM_BI := (Client:=Client,nObjectInstance:=10755);
	MalfunctionCode_042: FB_BACnetRM_MI := (Client:=Client,nObjectInstance:=10756);
	
	
	
	
	RoomTemp_042: FB_BACnetRM_AI := (Client:=Client,nObjectInstance:=10761);
	TempAdjust_042: FB_BACnetRM_AV := (Client:=Client,nObjectInstance:=10762);
	FilterSign_042: FB_BACnetRM_BI := (Client:=Client,nObjectInstance:=10763);
	FilterSignReset_042: FB_BACnetRM_BV := (Client:=Client,nObjectInstance:=10764);
	RemoteControlStart_042: FB_BACnetRM_BV := (Client:=Client,nObjectInstance:=10765);
	
	RemoteControlTempAdjust_042: FB_BACnetRM_BV := (Client:=Client,nObjectInstance:=10768);
	
	
	
	
	
	
	
	
	
	
	
	
	StartStopCommand_043: FB_BACnetRM_BO := (Client:=Client,nObjectInstance:=11009);
	StartStopStatus_043: FB_BACnetRM_BI := (Client:=Client,nObjectInstance:=11010);
	Alarm_043: FB_BACnetRM_BI := (Client:=Client,nObjectInstance:=11011);
	MalfunctionCode_043: FB_BACnetRM_MI := (Client:=Client,nObjectInstance:=11012);
	
	
	
	
	RoomTemp_043: FB_BACnetRM_AI := (Client:=Client,nObjectInstance:=11017);
	TempAdjust_043: FB_BACnetRM_AV := (Client:=Client,nObjectInstance:=11018);
	FilterSign_043: FB_BACnetRM_BI := (Client:=Client,nObjectInstance:=11019);
	FilterSignReset_043: FB_BACnetRM_BV := (Client:=Client,nObjectInstance:=11020);
	RemoteControlStart_043: FB_BACnetRM_BV := (Client:=Client,nObjectInstance:=11021);
	
	RemoteControlTempAdjust_043: FB_BACnetRM_BV := (Client:=Client,nObjectInstance:=11024);
	
	
	
	
	
	
	
	
	
	
	
	
	//StartStopCommand_044: FB_BACnetRM_BO := (Client:=Client,nObjectInstance:=11265);
	//StartStopStatus_044: FB_BACnetRM_BI := (Client:=Client,nObjectInstance:=11266);
	//Alarm_044: FB_BACnetRM_BI := (Client:=Client,nObjectInstance:=11267);
	//MalfunctionCode_044: FB_BACnetRM_MI := (Client:=Client,nObjectInstance:=11268);
	
	
	
	
	//RoomTemp_044: FB_BACnetRM_AI := (Client:=Client,nObjectInstance:=11273);
	//TempAdjust_044: FB_BACnetRM_AV := (Client:=Client,nObjectInstance:=11274);
	//FilterSign_044: FB_BACnetRM_BI := (Client:=Client,nObjectInstance:=11275);
	//FilterSignReset_044: FB_BACnetRM_BV := (Client:=Client,nObjectInstance:=11276);
	//RemoteControlStart_044: FB_BACnetRM_BV := (Client:=Client,nObjectInstance:=11277);
	//
	//RemoteControlTempAdjust_044: FB_BACnetRM_BV := (Client:=Client,nObjectInstance:=11280);
	
	//
	
	
	
	
	
	
	
	
	
	
	StartStopCommand_045: FB_BACnetRM_BO := (Client:=Client,nObjectInstance:=11521);
	StartStopStatus_045: FB_BACnetRM_BI := (Client:=Client,nObjectInstance:=11522);
	Alarm_045: FB_BACnetRM_BI := (Client:=Client,nObjectInstance:=11523);
	MalfunctionCode_045: FB_BACnetRM_MI := (Client:=Client,nObjectInstance:=11524);
	
	
	
	
	RoomTemp_045: FB_BACnetRM_AI := (Client:=Client,nObjectInstance:=11529);
	TempAdjust_045: FB_BACnetRM_AV := (Client:=Client,nObjectInstance:=11530);
	FilterSign_045: FB_BACnetRM_BI := (Client:=Client,nObjectInstance:=11531);
	FilterSignReset_045: FB_BACnetRM_BV := (Client:=Client,nObjectInstance:=11532);
	RemoteControlStart_045: FB_BACnetRM_BV := (Client:=Client,nObjectInstance:=11533);
	
	RemoteControlTempAdjust_045: FB_BACnetRM_BV := (Client:=Client,nObjectInstance:=11536);
	
	
	
	
	
	
	
	
	
	
	
	
	StartStopCommand_046: FB_BACnetRM_BO := (Client:=Client,nObjectInstance:=11777);
	StartStopStatus_046: FB_BACnetRM_BI := (Client:=Client,nObjectInstance:=11778);
	Alarm_046: FB_BACnetRM_BI := (Client:=Client,nObjectInstance:=11779);
	MalfunctionCode_046: FB_BACnetRM_MI := (Client:=Client,nObjectInstance:=11780);
	
	
	
	
	RoomTemp_046: FB_BACnetRM_AI := (Client:=Client,nObjectInstance:=11785);
	TempAdjust_046: FB_BACnetRM_AV := (Client:=Client,nObjectInstance:=11786);
	FilterSign_046: FB_BACnetRM_BI := (Client:=Client,nObjectInstance:=11787);
	FilterSignReset_046: FB_BACnetRM_BV := (Client:=Client,nObjectInstance:=11788);
	RemoteControlStart_046: FB_BACnetRM_BV := (Client:=Client,nObjectInstance:=11789);
	
	RemoteControlTempAdjust_046: FB_BACnetRM_BV := (Client:=Client,nObjectInstance:=11792);
	
	
	
	
	
	
	
	
	
	
	
	
	//StartStopCommand_048: FB_BACnetRM_BO := (Client:=Client,nObjectInstance:=12289);
	//StartStopStatus_048: FB_BACnetRM_BI := (Client:=Client,nObjectInstance:=12290);
	//Alarm_048: FB_BACnetRM_BI := (Client:=Client,nObjectInstance:=12291);
	//MalfunctionCode_048: FB_BACnetRM_MI := (Client:=Client,nObjectInstance:=12292);
	
	
	
	
	//RoomTemp_048: FB_BACnetRM_AI := (Client:=Client,nObjectInstance:=12297);
	//TempAdjust_048: FB_BACnetRM_AV := (Client:=Client,nObjectInstance:=12298);
	//FilterSign_048: FB_BACnetRM_BI := (Client:=Client,nObjectInstance:=12299);
	//FilterSignReset_048: FB_BACnetRM_BV := (Client:=Client,nObjectInstance:=12300);
	//RemoteControlStart_048: FB_BACnetRM_BV := (Client:=Client,nObjectInstance:=12301);
	//
	//RemoteControlTempAdjust_048: FB_BACnetRM_BV := (Client:=Client,nObjectInstance:=12304);
	
	//
	
	
	
	
	
	
	
	
	
	
	StartStopCommand_049: FB_BACnetRM_BO := (Client:=Client,nObjectInstance:=12545);
	StartStopStatus_049: FB_BACnetRM_BI := (Client:=Client,nObjectInstance:=12546);
	Alarm_049: FB_BACnetRM_BI := (Client:=Client,nObjectInstance:=12547);
	MalfunctionCode_049: FB_BACnetRM_MI := (Client:=Client,nObjectInstance:=12548);
	
	
	
	
	RoomTemp_049: FB_BACnetRM_AI := (Client:=Client,nObjectInstance:=12553);
	TempAdjust_049: FB_BACnetRM_AV := (Client:=Client,nObjectInstance:=12554);
	FilterSign_049: FB_BACnetRM_BI := (Client:=Client,nObjectInstance:=12555);
	FilterSignReset_049: FB_BACnetRM_BV := (Client:=Client,nObjectInstance:=12556);
	RemoteControlStart_049: FB_BACnetRM_BV := (Client:=Client,nObjectInstance:=12557);
	
	RemoteControlTempAdjust_049: FB_BACnetRM_BV := (Client:=Client,nObjectInstance:=12560);
	
	
	
	
	
	
	
	
	
	
	
	
	StartStopCommand_064: FB_BACnetRM_BO := (Client:=Client,nObjectInstance:=16385);
	StartStopStatus_064: FB_BACnetRM_BI := (Client:=Client,nObjectInstance:=16386);
	Alarm_064: FB_BACnetRM_BI := (Client:=Client,nObjectInstance:=16387);
	MalfunctionCode_064: FB_BACnetRM_MI := (Client:=Client,nObjectInstance:=16388);
	
	
	
	
	RoomTemp_064: FB_BACnetRM_AI := (Client:=Client,nObjectInstance:=16393);
	TempAdjust_064: FB_BACnetRM_AV := (Client:=Client,nObjectInstance:=16394);
	FilterSign_064: FB_BACnetRM_BI := (Client:=Client,nObjectInstance:=16395);
	FilterSignReset_064: FB_BACnetRM_BV := (Client:=Client,nObjectInstance:=16396);
	RemoteControlStart_064: FB_BACnetRM_BV := (Client:=Client,nObjectInstance:=16397);
	
	RemoteControlTempAdjust_064: FB_BACnetRM_BV := (Client:=Client,nObjectInstance:=16400);
	
	
	
	
	
	
	
	
	
	
	
	
	StartStopCommand_065: FB_BACnetRM_BO := (Client:=Client,nObjectInstance:=16641);
	StartStopStatus_065: FB_BACnetRM_BI := (Client:=Client,nObjectInstance:=16642);
	Alarm_065: FB_BACnetRM_BI := (Client:=Client,nObjectInstance:=16643);
	MalfunctionCode_065: FB_BACnetRM_MI := (Client:=Client,nObjectInstance:=16644);
	
	
	
	
	RoomTemp_065: FB_BACnetRM_AI := (Client:=Client,nObjectInstance:=16649);
	TempAdjust_065: FB_BACnetRM_AV := (Client:=Client,nObjectInstance:=16650);
	FilterSign_065: FB_BACnetRM_BI := (Client:=Client,nObjectInstance:=16651);
	FilterSignReset_065: FB_BACnetRM_BV := (Client:=Client,nObjectInstance:=16652);
	RemoteControlStart_065: FB_BACnetRM_BV := (Client:=Client,nObjectInstance:=16653);
	
	RemoteControlTempAdjust_065: FB_BACnetRM_BV := (Client:=Client,nObjectInstance:=16656);
	
	
	
	
	
	
	
	
	
	
	
	
	StartStopCommand_066: FB_BACnetRM_BO := (Client:=Client,nObjectInstance:=16897);
	StartStopStatus_066: FB_BACnetRM_BI := (Client:=Client,nObjectInstance:=16898);
	Alarm_066: FB_BACnetRM_BI := (Client:=Client,nObjectInstance:=16899);
	MalfunctionCode_066: FB_BACnetRM_MI := (Client:=Client,nObjectInstance:=16900);
	
	
	
	
	RoomTemp_066: FB_BACnetRM_AI := (Client:=Client,nObjectInstance:=16905);
	TempAdjust_066: FB_BACnetRM_AV := (Client:=Client,nObjectInstance:=16906);
	FilterSign_066: FB_BACnetRM_BI := (Client:=Client,nObjectInstance:=16907);
	FilterSignReset_066: FB_BACnetRM_BV := (Client:=Client,nObjectInstance:=16908);
	RemoteControlStart_066: FB_BACnetRM_BV := (Client:=Client,nObjectInstance:=16909);
	
	RemoteControlTempAdjust_066: FB_BACnetRM_BV := (Client:=Client,nObjectInstance:=16912);
	
	
	
	
	
	
	
	
	
	
	
	
	StartStopCommand_067: FB_BACnetRM_BO := (Client:=Client,nObjectInstance:=17153);
	StartStopStatus_067: FB_BACnetRM_BI := (Client:=Client,nObjectInstance:=17154);
	Alarm_067: FB_BACnetRM_BI := (Client:=Client,nObjectInstance:=17155);
	MalfunctionCode_067: FB_BACnetRM_MI := (Client:=Client,nObjectInstance:=17156);
	
	
	
	
	RoomTemp_067: FB_BACnetRM_AI := (Client:=Client,nObjectInstance:=17161);
	TempAdjust_067: FB_BACnetRM_AV := (Client:=Client,nObjectInstance:=17162);
	FilterSign_067: FB_BACnetRM_BI := (Client:=Client,nObjectInstance:=17163);
	FilterSignReset_067: FB_BACnetRM_BV := (Client:=Client,nObjectInstance:=17164);
	RemoteControlStart_067: FB_BACnetRM_BV := (Client:=Client,nObjectInstance:=17165);
	
	RemoteControlTempAdjust_067: FB_BACnetRM_BV := (Client:=Client,nObjectInstance:=17168);
	
	
	
	
	
	
	
	
	
	
	
	
	StartStopCommand_068: FB_BACnetRM_BO := (Client:=Client,nObjectInstance:=17409);
	StartStopStatus_068: FB_BACnetRM_BI := (Client:=Client,nObjectInstance:=17410);
	Alarm_068: FB_BACnetRM_BI := (Client:=Client,nObjectInstance:=17411);
	MalfunctionCode_068: FB_BACnetRM_MI := (Client:=Client,nObjectInstance:=17412);
	
	
	
	
	RoomTemp_068: FB_BACnetRM_AI := (Client:=Client,nObjectInstance:=17417);
	TempAdjust_068: FB_BACnetRM_AV := (Client:=Client,nObjectInstance:=17418);
	FilterSign_068: FB_BACnetRM_BI := (Client:=Client,nObjectInstance:=17419);
	FilterSignReset_068: FB_BACnetRM_BV := (Client:=Client,nObjectInstance:=17420);
	RemoteControlStart_068: FB_BACnetRM_BV := (Client:=Client,nObjectInstance:=17421);
	
	RemoteControlTempAdjust_068: FB_BACnetRM_BV := (Client:=Client,nObjectInstance:=17424);
	
	
	
	
	
	
	
	
	
	
	
	
	StartStopCommand_069: FB_BACnetRM_BO := (Client:=Client,nObjectInstance:=17665);
	StartStopStatus_069: FB_BACnetRM_BI := (Client:=Client,nObjectInstance:=17666);
	Alarm_069: FB_BACnetRM_BI := (Client:=Client,nObjectInstance:=17667);
	MalfunctionCode_069: FB_BACnetRM_MI := (Client:=Client,nObjectInstance:=17668);
	
	
	
	
	RoomTemp_069: FB_BACnetRM_AI := (Client:=Client,nObjectInstance:=17673);
	TempAdjust_069: FB_BACnetRM_AV := (Client:=Client,nObjectInstance:=17674);
	FilterSign_069: FB_BACnetRM_BI := (Client:=Client,nObjectInstance:=17675);
	FilterSignReset_069: FB_BACnetRM_BV := (Client:=Client,nObjectInstance:=17676);
	RemoteControlStart_069: FB_BACnetRM_BV := (Client:=Client,nObjectInstance:=17677);
	
	RemoteControlTempAdjust_069: FB_BACnetRM_BV := (Client:=Client,nObjectInstance:=17680);
	
	
	
	
	
	
	
	
	
	
	
	
	StartStopCommand_070: FB_BACnetRM_BO := (Client:=Client,nObjectInstance:=17921);
	StartStopStatus_070: FB_BACnetRM_BI := (Client:=Client,nObjectInstance:=17922);
	Alarm_070: FB_BACnetRM_BI := (Client:=Client,nObjectInstance:=17923);
	MalfunctionCode_070: FB_BACnetRM_MI := (Client:=Client,nObjectInstance:=17924);
	
	
	
	
	RoomTemp_070: FB_BACnetRM_AI := (Client:=Client,nObjectInstance:=17929);
	TempAdjust_070: FB_BACnetRM_AV := (Client:=Client,nObjectInstance:=17930);
	FilterSign_070: FB_BACnetRM_BI := (Client:=Client,nObjectInstance:=17931);
	FilterSignReset_070: FB_BACnetRM_BV := (Client:=Client,nObjectInstance:=17932);
	RemoteControlStart_070: FB_BACnetRM_BV := (Client:=Client,nObjectInstance:=17933);
	
	RemoteControlTempAdjust_070: FB_BACnetRM_BV := (Client:=Client,nObjectInstance:=17936);
	
	
	
	
	
	
	
	
	
	
	
	
	StartStopCommand_071: FB_BACnetRM_BO := (Client:=Client,nObjectInstance:=18177);
	StartStopStatus_071: FB_BACnetRM_BI := (Client:=Client,nObjectInstance:=18178);
	Alarm_071: FB_BACnetRM_BI := (Client:=Client,nObjectInstance:=18179);
	MalfunctionCode_071: FB_BACnetRM_MI := (Client:=Client,nObjectInstance:=18180);
	
	
	
	
	RoomTemp_071: FB_BACnetRM_AI := (Client:=Client,nObjectInstance:=18185);
	TempAdjust_071: FB_BACnetRM_AV := (Client:=Client,nObjectInstance:=18186);
	FilterSign_071: FB_BACnetRM_BI := (Client:=Client,nObjectInstance:=18187);
	FilterSignReset_071: FB_BACnetRM_BV := (Client:=Client,nObjectInstance:=18188);
	RemoteControlStart_071: FB_BACnetRM_BV := (Client:=Client,nObjectInstance:=18189);
	
	RemoteControlTempAdjust_071: FB_BACnetRM_BV := (Client:=Client,nObjectInstance:=18192);
	
	
	
	
	
	
	
	
	
	
	
	
	StartStopCommand_072: FB_BACnetRM_BO := (Client:=Client,nObjectInstance:=18433);
	StartStopStatus_072: FB_BACnetRM_BI := (Client:=Client,nObjectInstance:=18434);
	Alarm_072: FB_BACnetRM_BI := (Client:=Client,nObjectInstance:=18435);
	MalfunctionCode_072: FB_BACnetRM_MI := (Client:=Client,nObjectInstance:=18436);
	
	
	
	
	RoomTemp_072: FB_BACnetRM_AI := (Client:=Client,nObjectInstance:=18441);
	TempAdjust_072: FB_BACnetRM_AV := (Client:=Client,nObjectInstance:=18442);
	FilterSign_072: FB_BACnetRM_BI := (Client:=Client,nObjectInstance:=18443);
	FilterSignReset_072: FB_BACnetRM_BV := (Client:=Client,nObjectInstance:=18444);
	RemoteControlStart_072: FB_BACnetRM_BV := (Client:=Client,nObjectInstance:=18445);
	
	RemoteControlTempAdjust_072: FB_BACnetRM_BV := (Client:=Client,nObjectInstance:=18448);
	
	
	
	
	
	
	
	
	
	
	
	
	StartStopCommand_073: FB_BACnetRM_BO := (Client:=Client,nObjectInstance:=18689);
	StartStopStatus_073: FB_BACnetRM_BI := (Client:=Client,nObjectInstance:=18690);
	Alarm_073: FB_BACnetRM_BI := (Client:=Client,nObjectInstance:=18691);
	MalfunctionCode_073: FB_BACnetRM_MI := (Client:=Client,nObjectInstance:=18692);
	
	
	
	
	RoomTemp_073: FB_BACnetRM_AI := (Client:=Client,nObjectInstance:=18697);
	TempAdjust_073: FB_BACnetRM_AV := (Client:=Client,nObjectInstance:=18698);
	FilterSign_073: FB_BACnetRM_BI := (Client:=Client,nObjectInstance:=18699);
	FilterSignReset_073: FB_BACnetRM_BV := (Client:=Client,nObjectInstance:=18700);
	RemoteControlStart_073: FB_BACnetRM_BV := (Client:=Client,nObjectInstance:=18701);
	
	RemoteControlTempAdjust_073: FB_BACnetRM_BV := (Client:=Client,nObjectInstance:=18704);
	
	
	
	
	
	
	
	
	
	
	
	
	StartStopCommand_074: FB_BACnetRM_BO := (Client:=Client,nObjectInstance:=18945);
	StartStopStatus_074: FB_BACnetRM_BI := (Client:=Client,nObjectInstance:=18946);
	Alarm_074: FB_BACnetRM_BI := (Client:=Client,nObjectInstance:=18947);
	MalfunctionCode_074: FB_BACnetRM_MI := (Client:=Client,nObjectInstance:=18948);
	
	
	
	
	RoomTemp_074: FB_BACnetRM_AI := (Client:=Client,nObjectInstance:=18953);
	TempAdjust_074: FB_BACnetRM_AV := (Client:=Client,nObjectInstance:=18954);
	FilterSign_074: FB_BACnetRM_BI := (Client:=Client,nObjectInstance:=18955);
	FilterSignReset_074: FB_BACnetRM_BV := (Client:=Client,nObjectInstance:=18956);
	RemoteControlStart_074: FB_BACnetRM_BV := (Client:=Client,nObjectInstance:=18957);
	
	RemoteControlTempAdjust_074: FB_BACnetRM_BV := (Client:=Client,nObjectInstance:=18960);
	
	
	
	
	
	
	
	
	
	
	
	
	StartStopCommand_075: FB_BACnetRM_BO := (Client:=Client,nObjectInstance:=19201);
	StartStopStatus_075: FB_BACnetRM_BI := (Client:=Client,nObjectInstance:=19202);
	Alarm_075: FB_BACnetRM_BI := (Client:=Client,nObjectInstance:=19203);
	MalfunctionCode_075: FB_BACnetRM_MI := (Client:=Client,nObjectInstance:=19204);
	
	
	
	
	RoomTemp_075: FB_BACnetRM_AI := (Client:=Client,nObjectInstance:=19209);
	TempAdjust_075: FB_BACnetRM_AV := (Client:=Client,nObjectInstance:=19210);
	FilterSign_075: FB_BACnetRM_BI := (Client:=Client,nObjectInstance:=19211);
	FilterSignReset_075: FB_BACnetRM_BV := (Client:=Client,nObjectInstance:=19212);
	RemoteControlStart_075: FB_BACnetRM_BV := (Client:=Client,nObjectInstance:=19213);
	
	RemoteControlTempAdjust_075: FB_BACnetRM_BV := (Client:=Client,nObjectInstance:=19216);
	
	
	
	
	
	
	
	
	
	
	
	
	StartStopCommand_076: FB_BACnetRM_BO := (Client:=Client,nObjectInstance:=19457);
	StartStopStatus_076: FB_BACnetRM_BI := (Client:=Client,nObjectInstance:=19458);
	Alarm_076: FB_BACnetRM_BI := (Client:=Client,nObjectInstance:=19459);
	MalfunctionCode_076: FB_BACnetRM_MI := (Client:=Client,nObjectInstance:=19460);
	
	
	
	
	RoomTemp_076: FB_BACnetRM_AI := (Client:=Client,nObjectInstance:=19465);
	TempAdjust_076: FB_BACnetRM_AV := (Client:=Client,nObjectInstance:=19466);
	FilterSign_076: FB_BACnetRM_BI := (Client:=Client,nObjectInstance:=19467);
	FilterSignReset_076: FB_BACnetRM_BV := (Client:=Client,nObjectInstance:=19468);
	RemoteControlStart_076: FB_BACnetRM_BV := (Client:=Client,nObjectInstance:=19469);
	
	RemoteControlTempAdjust_076: FB_BACnetRM_BV := (Client:=Client,nObjectInstance:=19472);
	
	
	
	
	
	
	
	
	
	
	
	
	StartStopCommand_077: FB_BACnetRM_BO := (Client:=Client,nObjectInstance:=19713);
	StartStopStatus_077: FB_BACnetRM_BI := (Client:=Client,nObjectInstance:=19714);
	Alarm_077: FB_BACnetRM_BI := (Client:=Client,nObjectInstance:=19715);
	MalfunctionCode_077: FB_BACnetRM_MI := (Client:=Client,nObjectInstance:=19716);
	
	
	
	
	RoomTemp_077: FB_BACnetRM_AI := (Client:=Client,nObjectInstance:=19721);
	TempAdjust_077: FB_BACnetRM_AV := (Client:=Client,nObjectInstance:=19722);
	FilterSign_077: FB_BACnetRM_BI := (Client:=Client,nObjectInstance:=19723);
	FilterSignReset_077: FB_BACnetRM_BV := (Client:=Client,nObjectInstance:=19724);
	RemoteControlStart_077: FB_BACnetRM_BV := (Client:=Client,nObjectInstance:=19725);
	
	RemoteControlTempAdjust_077: FB_BACnetRM_BV := (Client:=Client,nObjectInstance:=19728);
	
	
	
	
	
	
	
	
	
	
	
	
	StartStopCommand_078: FB_BACnetRM_BO := (Client:=Client,nObjectInstance:=19969);
	StartStopStatus_078: FB_BACnetRM_BI := (Client:=Client,nObjectInstance:=19970);
	Alarm_078: FB_BACnetRM_BI := (Client:=Client,nObjectInstance:=19971);
	MalfunctionCode_078: FB_BACnetRM_MI := (Client:=Client,nObjectInstance:=19972);
	
	
	
	
	RoomTemp_078: FB_BACnetRM_AI := (Client:=Client,nObjectInstance:=19977);
	TempAdjust_078: FB_BACnetRM_AV := (Client:=Client,nObjectInstance:=19978);
	FilterSign_078: FB_BACnetRM_BI := (Client:=Client,nObjectInstance:=19979);
	FilterSignReset_078: FB_BACnetRM_BV := (Client:=Client,nObjectInstance:=19980);
	RemoteControlStart_078: FB_BACnetRM_BV := (Client:=Client,nObjectInstance:=19981);
	
	RemoteControlTempAdjust_078: FB_BACnetRM_BV := (Client:=Client,nObjectInstance:=19984);
	
	
	
	
	
	
	
	
	
	
	
	
	StartStopCommand_079: FB_BACnetRM_BO := (Client:=Client,nObjectInstance:=20225);
	StartStopStatus_079: FB_BACnetRM_BI := (Client:=Client,nObjectInstance:=20226);
	Alarm_079: FB_BACnetRM_BI := (Client:=Client,nObjectInstance:=20227);
	MalfunctionCode_079: FB_BACnetRM_MI := (Client:=Client,nObjectInstance:=20228);
	
	
	
	
	RoomTemp_079: FB_BACnetRM_AI := (Client:=Client,nObjectInstance:=20233);
	TempAdjust_079: FB_BACnetRM_AV := (Client:=Client,nObjectInstance:=20234);
	FilterSign_079: FB_BACnetRM_BI := (Client:=Client,nObjectInstance:=20235);
	FilterSignReset_079: FB_BACnetRM_BV := (Client:=Client,nObjectInstance:=20236);
	RemoteControlStart_079: FB_BACnetRM_BV := (Client:=Client,nObjectInstance:=20237);
	
	RemoteControlTempAdjust_079: FB_BACnetRM_BV := (Client:=Client,nObjectInstance:=20240);
	
	
	
	
	
	
	
	
	
	
	
	
	StartStopCommand_080: FB_BACnetRM_BO := (Client:=Client,nObjectInstance:=20481);
	StartStopStatus_080: FB_BACnetRM_BI := (Client:=Client,nObjectInstance:=20482);
	Alarm_080: FB_BACnetRM_BI := (Client:=Client,nObjectInstance:=20483);
	MalfunctionCode_080: FB_BACnetRM_MI := (Client:=Client,nObjectInstance:=20484);
	
	
	
	
	RoomTemp_080: FB_BACnetRM_AI := (Client:=Client,nObjectInstance:=20489);
	TempAdjust_080: FB_BACnetRM_AV := (Client:=Client,nObjectInstance:=20490);
	FilterSign_080: FB_BACnetRM_BI := (Client:=Client,nObjectInstance:=20491);
	FilterSignReset_080: FB_BACnetRM_BV := (Client:=Client,nObjectInstance:=20492);
	RemoteControlStart_080: FB_BACnetRM_BV := (Client:=Client,nObjectInstance:=20493);
	
	RemoteControlTempAdjust_080: FB_BACnetRM_BV := (Client:=Client,nObjectInstance:=20496);
	
	
	
	
	
	
	
	
	
	
	
	
	StartStopCommand_081: FB_BACnetRM_BO := (Client:=Client,nObjectInstance:=20737);
	StartStopStatus_081: FB_BACnetRM_BI := (Client:=Client,nObjectInstance:=20738);
	Alarm_081: FB_BACnetRM_BI := (Client:=Client,nObjectInstance:=20739);
	MalfunctionCode_081: FB_BACnetRM_MI := (Client:=Client,nObjectInstance:=20740);
	
	
	
	
	RoomTemp_081: FB_BACnetRM_AI := (Client:=Client,nObjectInstance:=20745);
	TempAdjust_081: FB_BACnetRM_AV := (Client:=Client,nObjectInstance:=20746);
	FilterSign_081: FB_BACnetRM_BI := (Client:=Client,nObjectInstance:=20747);
	FilterSignReset_081: FB_BACnetRM_BV := (Client:=Client,nObjectInstance:=20748);
	RemoteControlStart_081: FB_BACnetRM_BV := (Client:=Client,nObjectInstance:=20749);
	
	RemoteControlTempAdjust_081: FB_BACnetRM_BV := (Client:=Client,nObjectInstance:=20752);
	
	
	
	
	
	
	
	
	
	
	
	
	StartStopCommand_082: FB_BACnetRM_BO := (Client:=Client,nObjectInstance:=20993);
	StartStopStatus_082: FB_BACnetRM_BI := (Client:=Client,nObjectInstance:=20994);
	Alarm_082: FB_BACnetRM_BI := (Client:=Client,nObjectInstance:=20995);
	MalfunctionCode_082: FB_BACnetRM_MI := (Client:=Client,nObjectInstance:=20996);
	
	
	
	
	RoomTemp_082: FB_BACnetRM_AI := (Client:=Client,nObjectInstance:=21001);
	TempAdjust_082: FB_BACnetRM_AV := (Client:=Client,nObjectInstance:=21002);
	FilterSign_082: FB_BACnetRM_BI := (Client:=Client,nObjectInstance:=21003);
	FilterSignReset_082: FB_BACnetRM_BV := (Client:=Client,nObjectInstance:=21004);
	RemoteControlStart_082: FB_BACnetRM_BV := (Client:=Client,nObjectInstance:=21005);
	
	RemoteControlTempAdjust_082: FB_BACnetRM_BV := (Client:=Client,nObjectInstance:=21008);
	
	
	
	
	
	
	
	
	
	
	
	
	StartStopCommand_083: FB_BACnetRM_BO := (Client:=Client,nObjectInstance:=21249);
	StartStopStatus_083: FB_BACnetRM_BI := (Client:=Client,nObjectInstance:=21250);
	Alarm_083: FB_BACnetRM_BI := (Client:=Client,nObjectInstance:=21251);
	MalfunctionCode_083: FB_BACnetRM_MI := (Client:=Client,nObjectInstance:=21252);
	
	
	
	
	RoomTemp_083: FB_BACnetRM_AI := (Client:=Client,nObjectInstance:=21257);
	TempAdjust_083: FB_BACnetRM_AV := (Client:=Client,nObjectInstance:=21258);
	FilterSign_083: FB_BACnetRM_BI := (Client:=Client,nObjectInstance:=21259);
	FilterSignReset_083: FB_BACnetRM_BV := (Client:=Client,nObjectInstance:=21260);
	RemoteControlStart_083: FB_BACnetRM_BV := (Client:=Client,nObjectInstance:=21261);
	
	RemoteControlTempAdjust_083: FB_BACnetRM_BV := (Client:=Client,nObjectInstance:=21264);
	
	
	
	
	
	
	
	
	
	
	
	
	StartStopCommand_084: FB_BACnetRM_BO := (Client:=Client,nObjectInstance:=21505);
	StartStopStatus_084: FB_BACnetRM_BI := (Client:=Client,nObjectInstance:=21506);
	Alarm_084: FB_BACnetRM_BI := (Client:=Client,nObjectInstance:=21507);
	MalfunctionCode_084: FB_BACnetRM_MI := (Client:=Client,nObjectInstance:=21508);
	
	
	
	
	RoomTemp_084: FB_BACnetRM_AI := (Client:=Client,nObjectInstance:=21513);
	TempAdjust_084: FB_BACnetRM_AV := (Client:=Client,nObjectInstance:=21514);
	FilterSign_084: FB_BACnetRM_BI := (Client:=Client,nObjectInstance:=21515);
	FilterSignReset_084: FB_BACnetRM_BV := (Client:=Client,nObjectInstance:=21516);
	RemoteControlStart_084: FB_BACnetRM_BV := (Client:=Client,nObjectInstance:=21517);
	
	RemoteControlTempAdjust_084: FB_BACnetRM_BV := (Client:=Client,nObjectInstance:=21520);
	
	
	
	
	
	
	
	
	
	
	
	
